KUKA KRL program: MyProgram_171().src

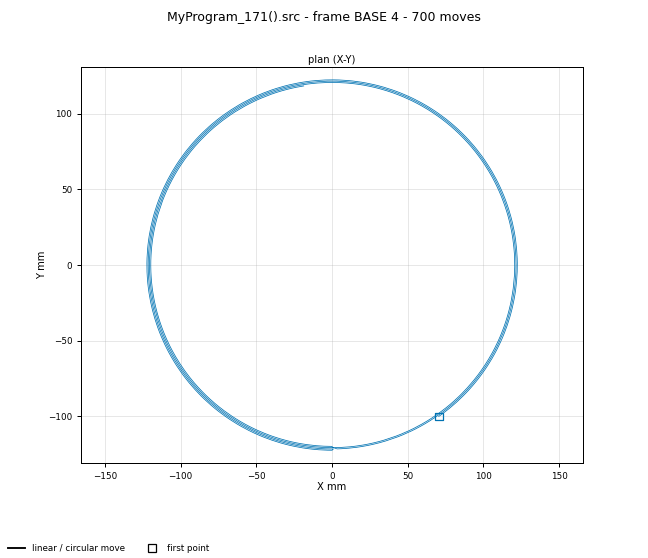
[picture p0: tool path of MyProgram_171().src in frame BASE 4, 700 of 700 moves have a stored position in this frame; points joined in program order, loops and branches not executed]
&ACCESS RVP
&REL 1
&PARAM TEMPLATE = C:\KRC\Roboter\Template\vorgabe
&PARAM EDITMASK = *
DEF MyProgram_171()
; ---- Setting reference (Base) ----
$BASE = BASE_DATA[4]

; --------------------------
; ---- Setting tool (TCP) ----
$TOOL = TOOL_DATA[3]
; --------------------------

$VEL.CP = VEL_APROX_PRINT
Startdeposition()
$VEL.CP = VEL_PRINT
LIN {X 70.4389,Y -100.0155,Z 128,A -58.0013,B 24.9588,C -1.4823,E1 25.0931,E2 504.1944} C_DIS
LIN {X 73.2543,Y -97.9697,Z 128,A -56.5791,B 24.9592,C -1.4754,E1 25.0962,E2 502.7935} C_DIS
LIN {X 75.6365,Y -96.1425,Z 128,A -55.0497,B 24.9587,C -1.4846,E1 25.0997,E2 501.248} C_DIS
LIN {X 77.6056,Y -94.5627,Z 128,A -53.6502,B 24.958,C -1.4981,E1 25.1027,E2 499.822} C_DIS
LIN {X 80.2629,Y -92.3154,Z 128,A -52.1799,B 24.9582,C -1.4939,E1 25.1058,E2 498.3674} C_DIS
LIN {X 82.1521,Y -90.6409,Z 128,A -50.8516,B 24.9576,C -1.504,E1 25.1086,E2 497.0206} C_DIS
LIN {X 84.6959,Y -88.2659,Z 128,A -49.3816,B 24.9579,C -1.4999,E1 25.1116,E2 495.5662} C_DIS
LIN {X 86.5007,Y -86.5007,Z 128,A -48.187,B 24.9577,C -1.5034,E1 25.1139,E2 494.3684} C_DIS
LIN {X 88.5975,Y -84.3518,Z 128,A -46.655,B 24.9571,C -1.5133,E1 25.1169,E2 492.8197} C_DIS
LIN {X 90.6409,Y -82.1521,Z 128,A -45.408,B 24.9573,C -1.5089,E1 25.1192,E2 491.5886} C_DIS
LIN {X 92.6297,Y -79.903,Z 128,A -43.8579,B 24.9567,C -1.5198,E1 25.1221,E2 490.0197} C_DIS
LIN {X 94.8636,Y -77.2344,Z 128,A -42.5892,B 24.9575,C -1.506,E1 25.1243,E2 488.7895} C_DIS
LIN {X 96.7305,Y -74.883,Z 128,A -41.1907,B 24.9573,C -1.5094,E1 25.1267,E2 487.3894} C_DIS
LIN {X 98.5391,Y -72.4866,Z 128,A -39.5927,B 24.9565,C -1.5229,E1 25.1294,E2 485.7672} C_DIS
LIN {X 100.8724,Y -69.2062,Z 128,A -37.5667,B 24.9558,C -1.5353,E1 25.1327,E2 483.7218} C_DIS
LIN {X 102.7986,Y -66.3077,Z 128,A -36.0983,B 24.956,C -1.5318,E1 25.1349,E2 482.269} C_DIS
LIN {X 104.3949,Y -63.7649,Z 128,A -34.9004,B 24.9564,C -1.5254,E1 25.1367,E2 481.0924} C_DIS
LIN {X 105.6902,Y -61.5981,Z 128,A -33.3738,B 24.9552,C -1.5463,E1 25.1389,E2 479.5245} C_DIS
LIN {X 107.3979,Y -58.5657,Z 128,A -31.9057,B 24.9554,C -1.5429,E1 25.1409,E2 478.0719} C_DIS
LIN {X 108.8029,Y -55.9124,Z 128,A -30.7084,B 24.9558,C -1.5366,E1 25.1424,E2 476.8958} C_DIS
LIN {X 110.1423,Y -53.2254,Z 128,A -29.1112,B 24.955,C -1.5505,E1 25.1444,E2 475.2744} C_DIS
LIN {X 111.219,Y -50.942,Z 128,A -27.9364,B 24.9548,C -1.5537,E1 25.1458,E2 474.0984} C_DIS
LIN {X 112.4356,Y -48.1972,Z 128,A -26.3877,B 24.9541,C -1.5653,E1 25.1475,E2 472.5308} C_DIS
LIN {X 113.7054,Y -45.1159,Z 128,A -25.1268,B 24.9547,C -1.555,E1 25.1488,E2 471.3013} C_DIS
LIN {X 114.8289,Y -42.1733,Z 128,A -23.5232,B 24.954,C -1.5661,E1 25.1504,E2 469.6803} C_DIS
LIN {X 115.6766,Y -39.7954,Z 128,A -22.3486,B 24.9538,C -1.5694,E1 25.1515,E2 468.5045} C_DIS
LIN {X 116.7599,Y -36.4881,Z 128,A -20.9292,B 24.9542,C -1.564,E1 25.1527,E2 467.106} C_DIS
LIN {X 117.4899,Y -34.0714,Z 128,A -19.5551,B 24.9534,C -1.5775,E1 25.1538,E2 465.708} C_DIS
LIN {X 118.4097,Y -30.715,Z 128,A -17.9362,B 24.9531,C -1.5822,E1 25.1549,E2 464.0872} C_DIS
LIN {X 119.1278,Y -27.7998,Z 128,A -16.7141,B 24.9534,C -1.5774,E1 25.1557,E2 462.8836} C_DIS
LIN {X 119.7741,Y -24.8679,Z 128,A -15.3426,B 24.9532,C -1.5802,E1 25.1566,E2 461.5134} C_DIS
LIN {X 120.2638,Y -22.3914,Z 128,A -13.9111,B 24.9522,C -1.5966,E1 25.1573,E2 460.0515} C_DIS
LIN {X 120.7771,Y -19.4332,Z 128,A -12.5721,B 24.9522,C -1.5978,E1 25.1579,E2 458.7176} C_DIS
LIN {X 121.2176,Y -16.4633,Z 128,A -11.1755,B 24.9519,C -1.6019,E1 25.1585,E2 457.3195} C_DIS
LIN {X 121.6349,Y -13.0082,Z 128,A -9.7568,B 24.9522,C -1.5966,E1 25.1589,E2 455.9219} C_DIS
LIN {X 121.8794,Y -10.4956,Z 128,A -8.3826,B 24.9514,C -1.6102,E1 25.1593,E2 454.5238} C_DIS
LIN {X 122.1266,Y -7.0242,Z 128,A -6.7638,B 24.9511,C -1.615,E1 25.1596,E2 452.9033} C_DIS
LIN {X 122.2476,Y -4.5026,Z 128,A -5.5896,B 24.9509,C -1.6184,E1 25.1597,E2 451.7279} C_DIS
LIN {X 122.3219,Y -1.3996,Z 128,A -4.203,B 24.9509,C -1.6198,E1 25.1597,E2 450.3464} C_DIS
LIN {X 122.3213,Y 1.5012,Z 128,A -2.645,B 24.9499,C -1.6343,E1 25.1597,E2 448.7633} C_DIS
LIN {X 122.2476,Y 4.5026,Z 128,A -1.4,B 24.9502,C -1.6307,E1 25.1597,E2 447.5342} C_DIS
LIN {X 122.068,Y 7.9782,Z 128,A 0.0188,B 24.9505,C -1.6254,E1 25.1594,E2 446.1364} C_DIS
LIN {X 121.8794,Y 10.4956,Z 128,A 1.5445,B 24.9492,C -1.6466,E1 25.1591,E2 444.5698} C_DIS
LIN {X 121.5295,Y 13.9582,Z 128,A 2.8121,B 24.95,C -1.6335,E1 25.1587,E2 443.3405} C_DIS
LIN {X 121.2176,Y 16.4633,Z 128,A 4.3379,B 24.9487,C -1.6547,E1 25.1581,E2 441.7738} C_DIS
LIN {X 120.7771,Y 19.4332,Z 128,A 5.7347,B 24.9484,C -1.6587,E1 25.1575,E2 440.3757} C_DIS
LIN {X 120.1591,Y 22.935,Z 128,A 7.2165,B 24.9487,C -1.6547,E1 25.1568,E2 438.912} C_DIS
LIN {X 119.5762,Y 25.8029,Z 128,A 8.3989,B 24.949,C -1.6495,E1 25.1561,E2 437.7487} C_DIS
LIN {X 119.0202,Y 28.2654,Z 128,A 9.7736,B 24.9482,C -1.6629,E1 25.1552,E2 436.3504} C_DIS
LIN {X 118.1661,Y 31.6392,Z 128,A 11.393,B 24.9479,C -1.6675,E1 25.1541,E2 434.7296} C_DIS
LIN {X 117.354,Y 34.5296,Z 128,A 12.7898,B 24.9477,C -1.6714,E1 25.153,E2 433.3317} C_DIS
LIN {X 116.6184,Y 36.9445,Z 128,A 13.9648,B 24.9475,C -1.6746,E1 25.152,E2 432.1558} C_DIS
LIN {X 115.6766,Y 39.7954,Z 128,A 15.362,B 24.9472,C -1.6784,E1 25.1508,E2 430.7575} C_DIS
LIN {X 114.4959,Y 43.0691,Z 128,A 16.9816,B 24.9469,C -1.6828,E1 25.1492,E2 429.1365} C_DIS
LIN {X 113.4044,Y 45.866,Z 128,A 18.379,B 24.9467,C -1.6865,E1 25.1478,E2 427.7382} C_DIS
LIN {X 112.2447,Y 48.6353,Z 128,A 19.7766,B 24.9465,C -1.6902,E1 25.1463,E2 426.3395} C_DIS
LIN {X 111.0173,Y 51.3753,Z 128,A 20.9741,B 24.9469,C -1.6838,E1 25.1449,E2 425.1636} C_DIS
LIN {X 109.723,Y 54.0843,Z 128,A 22.5719,B 24.946,C -1.6974,E1 25.1429,E2 423.5423} C_DIS
LIN {X 108.3627,Y 56.7608,Z 128,A 23.9696,B 24.9458,C -1.7009,E1 25.1411,E2 422.1436} C_DIS
LIN {X 106.9371,Y 59.403,Z 128,A 25.3677,B 24.9456,C -1.7044,E1 25.1393,E2 420.7446} C_DIS
LIN {X 105.6902,Y 61.5981,Z 128,A 26.5436,B 24.9454,C -1.7073,E1 25.1376,E2 419.568} C_DIS
LIN {X 103.8935,Y 64.5786,Z 128,A 28.1838,B 24.9451,C -1.7122,E1 25.1352,E2 417.9246} C_DIS
LIN {X 102.2598,Y 67.1355,Z 128,A 29.5683,B 24.9449,C -1.7141,E1 25.1331,E2 416.5425} C_DIS
LIN {X 100.8724,Y 69.2062,Z 128,A 30.7386,B 24.9447,C -1.7173,E1 25.1313,E2 415.3706} C_DIS
LIN {X 99.0399,Y 71.8026,Z 128,A 32.312,B 24.9442,C -1.7253,E1 25.1287,E2 413.7858} C_DIS
LIN {X 97.0634,Y 74.451,Z 128,A 33.5581,B 24.9449,C -1.7142,E1 25.1267,E2 412.5719} C_DIS
LIN {X 95.508,Y 76.4394,Z 128,A 34.9349,B 24.9441,C -1.7267,E1 25.1242,E2 411.1721} C_DIS
LIN {X 93.6033,Y 78.7602,Z 128,A 36.4861,B 24.9434,C -1.7372,E1 25.1214,E2 409.6032} C_DIS
LIN {X 90.6409,Y 82.1521,Z 128,A 38.585,B 24.9432,C -1.7416,E1 25.1175,E2 407.5033} C_DIS
LIN {X 88.2659,Y 84.6959,Z 128,A 40.0554,B 24.9434,C -1.7373,E1 25.1147,E2 406.0493} C_DIS
LIN {X 86.088,Y 86.9084,Z 128,A 41.4744,B 24.9434,C -1.7388,E1 25.112,E2 404.6329} C_DIS
LIN {X 82.9061,Y 89.9491,Z 128,A 43.555,B 24.943,C -1.744,E1 25.1077,E2 402.5484} C_DIS
LIN {X 80.6293,Y 91.9953,Z 128,A 44.9663,B 24.9429,C -1.7458,E1 25.1048,E2 401.1385} C_DIS
LIN {X 77.2344,Y 94.8636,Z 128,A 47.0559,B 24.9426,C -1.7503,E1 25.1003,E2 399.0465} C_DIS
LIN {X 74.883,Y 96.7305,Z 128,A 48.4567,B 24.9424,C -1.7526,E1 25.0972,E2 397.6453} C_DIS
LIN {X 72.4866,Y 98.5391,Z 128,A 49.8576,B 24.9423,C -1.7549,E1 25.0941,E2 396.2442} C_DIS
LIN {X 70.4389,Y 100.0155,Z 128,A 51.188,B 24.9417,C -1.7641,E1 25.091,E2 394.8966} C_DIS
LIN {X 67.5642,Y 101.9771,Z 128,A 52.6957,B 24.9419,C -1.7609,E1 25.0875,E2 393.4015} C_DIS
LIN {X 64.1733,Y 104.1467,Z 128,A 54.5393,B 24.9419,C -1.7618,E1 25.0832,E2 391.5618} C_DIS
LIN {X 61.1837,Y 105.9283,Z 128,A 56.1641,B 24.9417,C -1.764,E1 25.0793,E2 389.9367} C_DIS
LIN {X 58.5657,Y 107.3979,Z 128,A 57.566,B 24.9416,C -1.7657,E1 25.0758,E2 388.5347} C_DIS
LIN {X 55.9124,Y 108.8029,Z 128,A 58.9683,B 24.9415,C -1.7674,E1 25.0724,E2 387.1323} C_DIS
LIN {X 53.6561,Y 109.9353,Z 128,A 60.3,B 24.9409,C -1.7761,E1 25.069,E2 385.7836} C_DIS
LIN {X 50.7212,Y 111.3185,Z 128,A 61.7354,B 24.941,C -1.7738,E1 25.0654,E2 384.3572} C_DIS
LIN {X 47.7569,Y 112.6212,Z 128,A 63.1765,B 24.9412,C -1.7719,E1 25.0617,E2 382.9241} C_DIS
LIN {X 45.4234,Y 113.5846,Z 128,A 64.3564,B 24.9411,C -1.773,E1 25.0586,E2 381.7444} C_DIS
LIN {X 42.6222,Y 114.6651,Z 128,A 65.7597,B 24.9411,C -1.7742,E1 25.055,E2 380.3412} C_DIS
LIN {X 39.7954,Y 115.6766,Z 128,A 67.3158,B 24.9404,C -1.7826,E1 25.0508,E2 378.7683} C_DIS
LIN {X 36.4881,Y 116.7599,Z 128,A 68.664,B 24.9412,C -1.7705,E1 25.0473,E2 377.4512} C_DIS
LIN {X 34.0714,Y 117.4899,Z 128,A 69.9711,B 24.9408,C -1.7773,E1 25.0438,E2 376.1304} C_DIS
LIN {X 30.715,Y 118.4097,Z 128,A 71.3977,B 24.9414,C -1.7688,E1 25.04,E2 374.7263} C_DIS
LIN {X 27.7998,Y 119.1278,Z 128,A 72.8019,B 24.9414,C -1.7695,E1 25.0362,E2 373.3224} C_DIS
LIN {X 24.8679,Y 119.7741,Z 128,A 74.4081,B 24.9406,C -1.7796,E1 25.0318,E2 371.6942} C_DIS
LIN {X 22.3914,Y 120.2638,Z 128,A 75.5897,B 24.9406,C -1.7801,E1 25.0285,E2 370.513} C_DIS
LIN {X 19.4332,Y 120.7771,Z 128,A 76.9948,B 24.9406,C -1.7805,E1 25.0246,E2 369.1083} C_DIS
LIN {X 15.9894,Y 121.279,Z 128,A 78.4225,B 24.9412,C -1.7714,E1 25.0208,E2 367.7033} C_DIS
LIN {X 13.4835,Y 121.5851,Z 128,A 79.9588,B 24.9401,C -1.7882,E1 25.0164,E2 366.1283} C_DIS
LIN {X 10.1865,Y 121.9041,Z 128,A 81.356,B 24.9405,C -1.7812,E1 25.0126,E2 364.7487} C_DIS
LIN {X 7.0242,Y 122.1266,Z 128,A 82.8419,B 24.9405,C -1.7812,E1 25.0084,E2 363.2632} C_DIS
LIN {X 4.5026,Y 122.2476,Z 128,A 84.0246,B 24.9405,C -1.7812,E1 25.0051,E2 362.0811} C_DIS
LIN {X 1.0233,Y 122.3242,Z 128,A 85.4534,B 24.9412,C -1.7716,E1 25.0012,E2 360.6751} C_DIS
LIN {X -1.979,Y 122.3125,Z 128,A 87.0621,B 24.9406,C -1.7807,E1 24.9966,E2 359.0449} C_DIS
LIN {X -4.5026,Y 122.2476,Z 128,A 88.2453,B 24.9406,C -1.7803,E1 24.9933,E2 357.8624} C_DIS
LIN {X -7.9782,Y 122.068,Z 128,A 89.8768,B 24.9406,C -1.7798,E1 24.9888,E2 356.2317} C_DIS
LIN {X -10.4956,Y 121.8794,Z 128,A 91.0602,B 24.9406,C -1.7792,E1 24.9855,E2 355.049} C_DIS
LIN {X -13.9582,Y 121.5295,Z 128,A 92.5486,B 24.9412,C -1.7719,E1 24.9814,E2 353.5772} C_DIS
LIN {X -16.9365,Y 121.1504,Z 128,A 94.1004,B 24.9408,C -1.7777,E1 24.9771,E2 352.0104} C_DIS
LIN {X -19.9045,Y 120.6982,Z 128,A 95.5087,B 24.9408,C -1.7768,E1 24.9732,E2 350.603} C_DIS
LIN {X -22.8606,Y 120.1734,Z 128,A 96.7156,B 24.9415,C -1.7666,E1 24.9699,E2 349.4191} C_DIS
LIN {X -25.803,Y 119.5762,Z 128,A 98.2874,B 24.9411,C -1.7729,E1 24.9656,E2 347.8304} C_DIS
LIN {X -28.2654,Y 119.0202,Z 128,A 99.511,B 24.9411,C -1.7737,E1 24.9623,E2 346.6033} C_DIS
LIN {X -31.6392,Y 118.1661,Z 128,A 101.1446,B 24.9411,C -1.7722,E1 24.9578,E2 344.9708} C_DIS
LIN {X -34.5296,Y 117.354,Z 128,A 102.352,B 24.9418,C -1.7616,E1 24.9547,E2 343.7866} C_DIS
LIN {X -36.9445,Y 116.6184,Z 128,A 103.8928,B 24.9408,C -1.7766,E1 24.9505,E2 342.2076} C_DIS
LIN {X -39.7954,Y 115.6766,Z 128,A 105.1493,B 24.9414,C -1.768,E1 24.9472,E2 340.9692} C_DIS
LIN {X -43.0691,Y 114.4959,Z 128,A 106.7841,B 24.9415,C -1.7661,E1 24.9429,E2 339.3355} C_DIS
LIN {X -45.4234,Y 113.5846,Z 128,A 108.1235,B 24.9412,C -1.7715,E1 24.9394,E2 337.9803} C_DIS
LIN {X -48.6353,Y 112.2447,Z 128,A 109.6052,B 24.9418,C -1.7625,E1 24.9356,E2 336.5167} C_DIS
LIN {X -51.3753,Y 111.0173,Z 128,A 111.0161,B 24.9419,C -1.7605,E1 24.932,E2 335.1069} C_DIS
LIN {X -53.6561,Y 109.9353,Z 128,A 112.2025,B 24.942,C -1.7588,E1 24.9291,E2 333.9216} C_DIS
LIN {X -56.7608,Y 108.3627,Z 128,A 113.6359,B 24.9428,C -1.7473,E1 24.9256,E2 332.5117} C_DIS
LIN {X -58.9858,Y 107.1701,Z 128,A 115.1787,B 24.9419,C -1.7614,E1 24.9217,E2 330.931} C_DIS
LIN {X -61.5981,Y 105.6902,Z 128,A 116.5984,B 24.9419,C -1.7594,E1 24.9183,E2 329.5116} C_DIS
LIN {X -64.2066,Y 104.1259,Z 128,A 117.8506,B 24.9427,C -1.749,E1 24.9153,E2 328.2804} C_DIS
LIN {X -66.7099,Y 102.5404,Z 128,A 119.2609,B 24.9427,C -1.7474,E1 24.912,E2 326.8695} C_DIS
LIN {X -69.5986,Y 100.5996,Z 128,A 120.6954,B 24.9436,C -1.7354,E1 24.9087,E2 325.4586} C_DIS
LIN {X -71.6609,Y 99.1436,Z 128,A 122.0858,B 24.9431,C -1.7422,E1 24.9055,E2 324.0472} C_DIS
LIN {X -74.0725,Y 97.3551,Z 128,A 123.4985,B 24.9433,C -1.7395,E1 24.9024,E2 322.6359} C_DIS
LIN {X -76.4394,Y 95.508,Z 128,A 125.0647,B 24.943,C -1.7436,E1 24.8989,E2 321.0542} C_DIS
LIN {X -79.124,Y 93.2934,Z 128,A 126.549,B 24.9437,C -1.7334,E1 24.8958,E2 319.5883} C_DIS
LIN {X -81.3897,Y 91.3235,Z 128,A 127.7595,B 24.9445,C -1.7215,E1 24.8933,E2 318.4013} C_DIS
LIN {X -83.6064,Y 89.2986,Z 128,A 129.1729,B 24.9447,C -1.7185,E1 24.8904,E2 316.9894} C_DIS
LIN {X -85.4327,Y 87.5557,Z 128,A 130.7185,B 24.9438,C -1.7317,E1 24.8872,E2 315.406} C_DIS
LIN {X -87.5735,Y 85.4142,Z 128,A 131.979,B 24.9445,C -1.7212,E1 24.8848,E2 314.1651} C_DIS
LIN {X -89.9491,Y 82.9061,Z 128,A 133.6167,B 24.9447,C -1.718,E1 24.8817,E2 312.5278} C_DIS
LIN {X -91.9566,Y 80.6737,Z 128,A 135.0309,B 24.9449,C -1.7148,E1 24.879,E2 311.1151} C_DIS
LIN {X -93.9087,Y 78.3927,Z 128,A 136.445,B 24.9451,C -1.7114,E1 24.8765,E2 309.7024} C_DIS
LIN {X -95.7506,Y 76.1323,Z 128,A 137.6524,B 24.9458,C -1.7008,E1 24.8744,E2 308.5146} C_DIS
LIN {X -97.4209,Y 73.9849,Z 128,A 139.2166,B 24.9452,C -1.7101,E1 24.8717,E2 306.9209} C_DIS
LIN {X -99.4212,Y 71.2719,Z 128,A 140.6881,B 24.9458,C -1.701,E1 24.8693,E2 305.4638} C_DIS
LIN {X -100.8724,Y 69.2062,Z 128,A 141.8779,B 24.946,C -1.698,E1 24.8674,E2 304.2753} C_DIS
LIN {X -102.7986,Y 66.3077,Z 128,A 143.315,B 24.9468,C -1.685,E1 24.8653,E2 302.8621} C_DIS
LIN {X -104.3949,Y 63.7649,Z 128,A 144.9327,B 24.9465,C -1.6902,E1 24.8628,E2 301.2238} C_DIS
LIN {X -105.6902,Y 61.5981,Z 128,A 146.1228,B 24.9467,C -1.687,E1 24.8612,E2 300.035} C_DIS
LIN {X -107.3979,Y 58.5657,Z 128,A 147.7629,B 24.9469,C -1.6827,E1 24.8589,E2 298.3967} C_DIS
LIN {X -108.5854,Y 56.3379,Z 128,A 148.9532,B 24.9471,C -1.6795,E1 24.8574,E2 297.2077} C_DIS
LIN {X -110.1423,Y 53.2254,Z 128,A 150.3908,B 24.948,C -1.6662,E1 24.8556,E2 295.794} C_DIS
LIN {X -111.219,Y 50.942,Z 128,A 151.7839,B 24.9476,C -1.6717,E1 24.854,E2 294.3801} C_DIS
LIN {X -112.4356,Y 48.1972,Z 128,A 153.1996,B 24.9479,C -1.6678,E1 24.8524,E2 292.9659} C_DIS
LIN {X -113.5846,Y 45.4234,Z 128,A 154.6152,B 24.9481,C -1.6638,E1 24.8509,E2 291.5519} C_DIS
LIN {X -114.6651,Y 42.6222,Z 128,A 156.0308,B 24.9484,C -1.6599,E1 24.8495,E2 290.1377} C_DIS
LIN {X -115.8293,Y 39.3425,Z 128,A 157.6716,B 24.9487,C -1.6552,E1 24.848,E2 288.4987} C_DIS
LIN {X -116.7599,Y 36.4881,Z 128,A 158.8849,B 24.9495,C -1.6424,E1 24.847,E2 287.3091} C_DIS
LIN {X -117.4899,Y 34.0714,Z 128,A 160.2783,B 24.9491,C -1.6477,E1 24.8459,E2 285.8948} C_DIS
LIN {X -118.4097,Y 30.715,Z 128,A 161.7167,B 24.95,C -1.6342,E1 24.8448,E2 284.4803} C_DIS
LIN {X -119.1278,Y 27.7998,Z 128,A 163.1324,B 24.9502,C -1.6301,E1 24.8439,E2 283.0662} C_DIS
LIN {X -119.7144,Y 25.1591,Z 128,A 164.5349,B 24.9502,C -1.6318,E1 24.8431,E2 281.6513} C_DIS
LIN {X -120.2638,Y 22.3914,Z 128,A 165.9425,B 24.9502,C -1.6313,E1 24.8423,E2 280.2367} C_DIS
LIN {X -120.7771,Y 19.4332,Z 128,A 167.5124,B 24.95,C -1.6338,E1 24.8416,E2 278.6513} C_DIS
LIN {X -121.279,Y 15.9894,Z 128,A 168.7971,B 24.9512,C -1.6135,E1 24.8411,E2 277.4074} C_DIS
LIN {X -121.6349,Y 13.0082,Z 128,A 170.4159,B 24.9509,C -1.6181,E1 24.8406,E2 275.7679} C_DIS
LIN {X -121.9175,Y 10.0192,Z 128,A 171.8018,B 24.9513,C -1.6127,E1 24.8403,E2 274.3868} C_DIS
LIN {X -122.1266,Y 7.0242,Z 128,A 173.2484,B 24.9514,C -1.6098,E1 24.84,E2 272.9382} C_DIS
LIN {X -122.2476,Y 4.5026,Z 128,A 174.4392,B 24.9517,C -1.6063,E1 24.8399,E2 271.7487} C_DIS
LIN {X -122.3233,Y 1.1863,Z 128,A 176.0133,B 24.9519,C -1.6021,E1 24.8398,E2 270.175} C_DIS
LIN {X -122.3125,Y -1.979,Z 128,A 177.4968,B 24.9522,C -1.5973,E1 24.8398,E2 268.694} C_DIS
LIN {X -122.2476,Y -4.5026,Z 128,A 178.6875,B 24.9524,C -1.5938,E1 24.8399,E2 267.5045} C_DIS
LIN {X -122.068,Y -7.9782,Z 128,A -179.6453,B 24.9526,C -1.5901,E1 24.8402,E2 265.836} C_DIS
LIN {X -121.7414,Y -11.9905,Z 128,A -177.6185,B 24.9526,C -1.5901,E1 24.8407,E2 263.797} C_DIS
LIN {X -121.3491,Y -15.4485,Z 128,A -176.1313,B 24.9533,C -1.5787,E1 24.8412,E2 262.3282} C_DIS
LIN {X -120.9334,Y -18.4219,Z 128,A -174.7152,B 24.9535,C -1.5747,E1 24.8418,E2 260.9134} C_DIS
LIN {X -120.4449,Y -21.3842,Z 128,A -173.2995,B 24.9538,C -1.5706,E1 24.8425,E2 259.4989} C_DIS
LIN {X -119.8927,Y -24.2902,Z 128,A -171.8914,B 24.954,C -1.5672,E1 24.8432,E2 258.0906} C_DIS
LIN {X -119.3581,Y -26.8028,Z 128,A -170.693,B 24.9542,C -1.5632,E1 24.8439,E2 256.8947} C_DIS
LIN {X -118.6644,Y -29.7239,Z 128,A -169.1237,B 24.9541,C -1.5659,E1 24.845,E2 255.3096} C_DIS
LIN {X -117.7689,Y -33.0869,Z 128,A -167.6366,B 24.9547,C -1.5547,E1 24.8461,E2 253.8408} C_DIS
LIN {X -117.063,Y -35.5107,Z 128,A -166.2925,B 24.9545,C -1.5581,E1 24.8472,E2 252.4808} C_DIS
LIN {X -116.0035,Y -38.8257,Z 128,A -165.0085,B 24.9557,C -1.538,E1 24.8482,E2 251.2373} C_DIS
LIN {X -115.1795,Y -41.2119,Z 128,A -163.4617,B 24.955,C -1.5504,E1 24.8497,E2 249.6521} C_DIS
LIN {X -113.9587,Y -44.4709,Z 128,A -162.1781,B 24.9561,C -1.5303,E1 24.8509,E2 248.4091} C_DIS
LIN {X -112.833,Y -47.2542,Z 128,A -160.5601,B 24.9558,C -1.5355,E1 24.8527,E2 246.7698} C_DIS
LIN {X -111.6394,Y -50.0091,Z 128,A -159.3475,B 24.9565,C -1.5229,E1 24.854,E2 245.5806} C_DIS
LIN {X -110.5854,Y -52.303,Z 128,A -157.8015,B 24.9558,C -1.5355,E1 24.8559,E2 243.996} C_DIS
LIN {X -109.2686,Y -55.0012,Z 128,A -156.5402,B 24.9564,C -1.5251,E1 24.8574,E2 242.7528} C_DIS
LIN {X -107.8859,Y -57.6662,Z 128,A -155.1256,B 24.9566,C -1.5216,E1 24.8593,E2 241.3391} C_DIS
LIN {X -106.2001,Y -60.7108,Z 128,A -153.4379,B 24.9567,C -1.5197,E1 24.8616,E2 239.6471} C_DIS
LIN {X -104.1467,Y -64.1733,Z 128,A -151.5897,B 24.9571,C -1.5129,E1 24.8643,E2 237.8054} C_DIS
LIN {X -102.5404,Y -66.7099,Z 128,A -150.022,B 24.9569,C -1.5164,E1 24.8666,E2 236.2214} C_DIS
LIN {X -100.5996,Y -69.5986,Z 128,A -148.7391,B 24.958,C -1.4968,E1 24.8686,E2 234.9789} C_DIS
LIN {X -99.1436,Y -71.6609,Z 128,A -147.1939,B 24.9573,C -1.51,E1 24.8712,E2 233.3949} C_DIS
LIN {X -97.0201,Y -74.5073,Z 128,A -145.6955,B 24.9579,C -1.4985,E1 24.8737,E2 231.9165} C_DIS
LIN {X -94.5627,Y -77.6056,Z 128,A -143.66,B 24.9577,C -1.5022,E1 24.8773,E2 229.8627} C_DIS
LIN {X -92.3154,Y -80.2629,Z 128,A -142.1753,B 24.9583,C -1.4919,E1 24.8799,E2 228.3958} C_DIS
LIN {X -90.6409,Y -82.1521,Z 128,A -140.8336,B 24.9581,C -1.4964,E1 24.8825,E2 227.0376} C_DIS
LIN {X -88.2659,Y -84.6959,Z 128,A -139.3492,B 24.9586,C -1.4862,E1 24.8853,E2 225.5708} C_DIS
LIN {X -86.5007,Y -86.5007,Z 128,A -138.1613,B 24.9587,C -1.4839,E1 24.8876,E2 224.3834} C_DIS
LIN {X -84.3518,Y -88.5975,Z 128,A -136.5954,B 24.9585,C -1.4881,E1 24.8908,E2 222.8009} C_DIS
LIN {X -81.8156,Y -90.9422,Z 128,A -135.315,B 24.9595,C -1.4696,E1 24.8934,E2 221.5594} C_DIS
LIN {X -79.903,Y -92.6297,Z 128,A -133.7708,B 24.9588,C -1.4831,E1 24.8967,E2 219.9772} C_DIS
LIN {X -77.2344,Y -94.8636,Z 128,A -132.4901,B 24.9598,C -1.4641,E1 24.8994,E2 218.7366} C_DIS
LIN {X -74.883,Y -96.7305,Z 128,A -130.8258,B 24.9593,C -1.4733,E1 24.9031,E2 217.0445} C_DIS
LIN {X -72.4866,Y -98.5391,Z 128,A -129.4643,B 24.9596,C -1.4687,E1 24.9061,E2 215.6889} C_DIS
LIN {X -70.4389,Y -100.0155,Z 128,A -128.2773,B 24.9596,C -1.4669,E1 24.9088,E2 214.5022} C_DIS
LIN {X -67.5642,Y -101.9771,Z 128,A -126.6415,B 24.9598,C -1.4645,E1 24.9126,E2 212.8667} C_DIS
LIN {X -65.0412,Y -103.6045,Z 128,A -125.2306,B 24.9599,C -1.4625,E1 24.9159,E2 211.4559} C_DIS
LIN {X -62.8904,Y -104.9264,Z 128,A -124.0444,B 24.96,C -1.4609,E1 24.9188,E2 210.2699} C_DIS
LIN {X -59.8792,Y -106.6712,Z 128,A -122.4094,B 24.9601,C -1.4588,E1 24.9227,E2 208.6351} C_DIS
LIN {X -57.2434,Y -108.1085,Z 128,A -120.9991,B 24.9602,C -1.4571,E1 24.9262,E2 207.2248} C_DIS
LIN {X -55.0012,Y -109.2686,Z 128,A -119.6604,B 24.9599,C -1.4628,E1 24.9296,E2 205.869} C_DIS
LIN {X -51.8698,Y -110.7871,Z 128,A -118.1491,B 24.9603,C -1.4554,E1 24.9334,E2 204.3715} C_DIS
LIN {X -48.1972,Y -112.4356,Z 128,A -116.1362,B 24.9601,C -1.4592,E1 24.9385,E2 202.3448} C_DIS
LIN {X -45.4234,Y -113.5846,Z 128,A -114.7346,B 24.9602,C -1.4575,E1 24.9422,E2 200.9441} C_DIS
LIN {X -42.1733,Y -114.8289,Z 128,A -113.2466,B 24.9606,C -1.4494,E1 24.946,E2 199.4722} C_DIS
LIN {X -39.7954,Y -115.6766,Z 128,A -112.0563,B 24.9606,C -1.4488,E1 24.9492,E2 198.2812} C_DIS
LIN {X -36.4881,Y -116.7599,Z 128,A -110.6306,B 24.9613,C -1.438,E1 24.9529,E2 196.8785} C_DIS
LIN {X -34.0714,Y -117.4899,Z 128,A -109.2449,B 24.9608,C -1.4466,E1 24.9567,E2 195.47} C_DIS
LIN {X -30.715,Y -118.4097,Z 128,A -107.6128,B 24.9608,C -1.4457,E1 24.9611,E2 193.8375} C_DIS
LIN {X -27.7998,Y -119.1278,Z 128,A -106.4066,B 24.9614,C -1.4356,E1 24.9643,E2 192.6537} C_DIS
LIN {X -24.8679,Y -119.7741,Z 128,A -104.9985,B 24.9614,C -1.435,E1 24.9681,E2 191.2453} C_DIS
LIN {X -21.906,Y -120.3511,Z 128,A -103.5905,B 24.9614,C -1.4342,E1 24.972,E2 189.8377} C_DIS
LIN {X -19.4332,Y -120.7771,Z 128,A -102.2066,B 24.961,C -1.4436,E1 24.9759,E2 188.4301} C_DIS
LIN {X -16.4633,Y -121.2176,Z 128,A -100.7996,B 24.961,C -1.4433,E1 24.9798,E2 187.0227} C_DIS
LIN {X -13.0082,Y -121.6349,Z 128,A -99.1438,B 24.961,C -1.4443,E1 24.9844,E2 185.3633} C_DIS
LIN {X -8.9992,Y -121.999,Z 128,A -97.1309,B 24.9606,C -1.4503,E1 24.99,E2 183.3354} C_DIS
LIN {X -5.525,Y -122.2036,Z 128,A -95.8548,B 24.9615,C -1.4336,E1 24.9935,E2 182.0986} C_DIS
LIN {X -3.0021,Y -122.2936,Z 128,A -94.3189,B 24.9606,C -1.4506,E1 24.9979,E2 180.5223} C_DIS
LIN {X 0,Y -122.3305,Z 128,A -92.9133,B 24.9606,C -1.4508,E1 25.0018,E2 179.1161} C_DIS
LIN {X 0,Y -122.3305,Z 128,A -92.9133,B 24.9606,C -1.4508,E1 25.0018,E2 179.1161} C_DIS
Enddeposition()
LIN {X 0.8564,Y -121.47,Z 128,A -92.5769,B 24.9599,C -1.4627,E1 25.0028,E2 178.7516} C_DIS
Startdeposition()
$VEL.CP = VEL_PRINT
LIN {X -0.9647,Y -121.4729,Z 128,A -94.2168,B 24.9619,C -1.4256,E1 24.998,E2 180.4793} C_DIS
LIN {X -4.555,Y -121.3929,Z 128,A -96.0357,B 24.9623,C -1.4195,E1 24.9929,E2 182.3129} C_DIS
LIN {X -9.0533,Y -121.1404,Z 128,A -98.2299,B 24.9624,C -1.4163,E1 24.9867,E2 184.5156} C_DIS
LIN {X -13.6853,Y -120.7041,Z 128,A -100.2672,B 24.962,C -1.4238,E1 24.9811,E2 186.5362} C_DIS
LIN {X -17.9499,Y -120.1444,Z 128,A -102.1563,B 24.9617,C -1.4307,E1 24.9759,E2 188.4105} C_DIS
LIN {X -23.0019,Y -119.279,Z 128,A -104.5486,B 24.9616,C -1.4326,E1 24.9694,E2 190.8004} C_DIS
LIN {X -25.7925,Y -118.7068,Z 128,A -106.0689,B 24.962,C -1.4251,E1 24.9651,E2 192.3404} C_DIS
LIN {X -29.1299,Y -117.9327,Z 128,A -107.5553,B 24.9616,C -1.4319,E1 24.9611,E2 193.8127} C_DIS
LIN {X -32.1278,Y -117.1519,Z 128,A -109.0894,B 24.9617,C -1.4295,E1 24.957,E2 195.3549} C_DIS
LIN {X -35.8702,Y -116.0599,Z 128,A -111.0253,B 24.9619,C -1.4263,E1 24.9518,E2 197.3015} C_DIS
LIN {X -38.6924,Y -115.1498,Z 128,A -112.4178,B 24.9619,C -1.4277,E1 24.9481,E2 198.6933} C_DIS
LIN {X -41.7788,Y -114.0663,Z 128,A -113.9264,B 24.9617,C -1.4307,E1 24.9441,E2 200.1979} C_DIS
LIN {X -45.5578,Y -112.6104,Z 128,A -115.8907,B 24.9617,C -1.4301,E1 24.939,E2 202.1678} C_DIS
LIN {X -49.3374,Y -111.008,Z 128,A -117.8037,B 24.9615,C -1.4332,E1 24.9341,E2 204.0778} C_DIS
LIN {X -52.4934,Y -109.5491,Z 128,A -119.3831,B 24.9613,C -1.4379,E1 24.9301,E2 205.6501} C_DIS
LIN {X -55.8126,Y -107.8975,Z 128,A -121.103,B 24.9611,C -1.4414,E1 24.9259,E2 207.3663} C_DIS
LIN {X -58.0544,Y -106.7064,Z 128,A -122.3071,B 24.9611,C -1.4428,E1 24.9229,E2 208.5706} C_DIS
LIN {X -60.7675,Y -105.1853,Z 128,A -123.8443,B 24.9611,C -1.4417,E1 24.9192,E2 210.1148} C_DIS
LIN {X -63.5715,Y -103.5159,Z 128,A -125.3187,B 24.9608,C -1.4469,E1 24.9156,E2 211.5815} C_DIS
LIN {X -66.1342,Y -101.898,Z 128,A -126.9367,B 24.9611,C -1.4407,E1 24.9118,E2 213.2194} C_DIS
LIN {X -69.9741,Y -99.301,Z 128,A -129.1106,B 24.9609,C -1.4449,E1 24.9068,E2 215.3906} C_DIS
LIN {X -73.0883,Y -97.0293,Z 128,A -130.7953,B 24.9604,C -1.4541,E1 24.9031,E2 217.0595} C_DIS
LIN {X -75.5152,Y -95.1529,Z 128,A -132.2867,B 24.9604,C -1.4547,E1 24.8998,E2 218.5548} C_DIS
LIN {X -78.2157,Y -92.9481,Z 128,A -133.8764,B 24.9601,C -1.4603,E1 24.8964,E2 220.1375} C_DIS
LIN {X -80.0842,Y -91.3407,Z 128,A -135.0356,B 24.9599,C -1.4627,E1 24.8939,E2 221.2953} C_DIS
LIN {X -82.2674,Y -89.3794,Z 128,A -136.5698,B 24.9601,C -1.4589,E1 24.8907,E2 222.8447} C_DIS
LIN {X -85.0049,Y -86.7813,Z 128,A -138.4181,B 24.9601,C -1.4597,E1 24.887,E2 224.699} C_DIS
LIN {X -87.6266,Y -84.132,Z 128,A -140.0981,B 24.9597,C -1.467,E1 24.8838,E2 226.3688} C_DIS
LIN {X -90.1201,Y -81.4571,Z 128,A -141.87,B 24.9596,C -1.4688,E1 24.8804,E2 228.1443} C_DIS
LIN {X -92.7192,Y -78.4848,Z 128,A -143.6139,B 24.9591,C -1.4783,E1 24.8772,E2 229.8734} C_DIS
LIN {X -94.7059,Y -76.0765,Z 128,A -145.0772,B 24.9588,C -1.4822,E1 24.8747,E2 231.3341} C_DIS
LIN {X -96.9086,Y -73.2489,Z 128,A -146.9191,B 24.959,C -1.4798,E1 24.8715,E2 233.1907} C_DIS
LIN {X -99.1588,Y -70.1734,Z 128,A -148.6115,B 24.9585,C -1.4889,E1 24.8688,E2 234.8697} C_DIS
LIN {X -100.9336,Y -67.597,Z 128,A -150.0543,B 24.9582,C -1.4941,E1 24.8665,E2 236.3071} C_DIS
LIN {X -102.5688,Y -65.0891,Z 128,A -151.4782,B 24.958,C -1.4973,E1 24.8644,E2 237.7306} C_DIS
LIN {X -104.2177,Y -62.4157,Z 128,A -153.2269,B 24.9584,C -1.4897,E1 24.8618,E2 239.5065} C_DIS
LIN {X -106.4782,Y -58.4752,Z 128,A -155.2855,B 24.9579,C -1.4992,E1 24.859,E2 241.5532} C_DIS
LIN {X -108.1197,Y -55.3778,Z 128,A -156.8253,B 24.9574,C -1.5087,E1 24.857,E2 243.0784} C_DIS
LIN {X -109.5034,Y -52.5887,Z 128,A -158.3584,B 24.9573,C -1.5101,E1 24.8551,E2 244.6165} C_DIS
LIN {X -110.8398,Y -49.7106,Z 128,A -159.8436,B 24.957,C -1.5149,E1 24.8534,E2 246.0985} C_DIS
LIN {X -112.4607,Y -45.9256,Z 128,A -161.7733,B 24.9566,C -1.5211,E1 24.8513,E2 248.024} C_DIS
LIN {X -113.6259,Y -42.9618,Z 128,A -163.4959,B 24.9569,C -1.5161,E1 24.8496,E2 249.7682} C_DIS
LIN {X -114.9148,Y -39.3893,Z 128,A -165.2066,B 24.9564,C -1.525,E1 24.848,E2 251.4676} C_DIS
LIN {X -116.068,Y -35.8442,Z 128,A -166.8746,B 24.9559,C -1.5342,E1 24.8466,E2 253.1231} C_DIS
LIN {X -116.9478,Y -32.8609,Z 128,A -168.5712,B 24.9562,C -1.5289,E1 24.8453,E2 254.8423} C_DIS
LIN {X -117.9614,Y -29.0123,Z 128,A -170.2234,B 24.9553,C -1.5444,E1 24.8442,E2 256.4672} C_DIS
LIN {X -118.6984,Y -25.831,Z 128,A -171.7654,B 24.955,C -1.5491,E1 24.8433,E2 258.0069} C_DIS
LIN {X -119.4275,Y -22.2279,Z 128,A -173.4713,B 24.9547,C -1.5558,E1 24.8423,E2 259.707} C_DIS
LIN {X -119.8705,Y -19.6908,Z 128,A -174.8571,B 24.9548,C -1.5524,E1 24.8417,E2 261.1092} C_DIS
LIN {X -120.4702,Y -15.6044,Z 128,A -176.6949,B 24.9542,C -1.5633,E1 24.841,E2 262.9319} C_DIS
LIN {X -120.8293,Y -12.5236,Z 128,A -178.1645,B 24.9539,C -1.5677,E1 24.8405,E2 264.3998} C_DIS
LIN {X -121.1484,Y -8.9531,Z 128,A 179.9828,B 24.954,C -1.5663,E1 24.8401,E2 266.2671} C_DIS
LIN {X -121.367,Y -5.1596,Z 128,A 178.3084,B 24.9534,C -1.5772,E1 24.8399,E2 267.9256} C_DIS
LIN {X -121.4616,Y -1.9319,Z 128,A 176.827,B 24.953,C -1.5839,E1 24.8398,E2 269.3998} C_DIS
LIN {X -121.4737,Y 0.8721,Z 128,A 175.4506,B 24.9529,C -1.5859,E1 24.8398,E2 270.7797} C_DIS
LIN {X -121.3942,Y 4.5248,Z 128,A 173.584,B 24.9529,C -1.5854,E1 24.84,E2 272.6587} C_DIS
LIN {X -121.2009,Y 8.1796,Z 128,A 171.9423,B 24.9523,C -1.5947,E1 24.8402,E2 274.2882} C_DIS
LIN {X -120.9642,Y 11.1457,Z 128,A 170.5873,B 24.952,C -1.6014,E1 24.8406,E2 275.6355} C_DIS
LIN {X -120.6256,Y 14.3549,Z 128,A 169.0419,B 24.9517,C -1.6053,E1 24.841,E2 277.1807} C_DIS
LIN {X -120.2475,Y 17.2368,Z 128,A 167.6268,B 24.9516,C -1.6079,E1 24.8416,E2 278.598} C_DIS
LIN {X -119.6264,Y 21.1241,Z 128,A 165.7103,B 24.9513,C -1.6114,E1 24.8425,E2 280.5175} C_DIS
LIN {X -118.9252,Y 24.7684,Z 128,A 163.8807,B 24.9513,C -1.6138,E1 24.8435,E2 282.3524} C_DIS
LIN {X -118.0544,Y 28.6313,Z 128,A 162.0982,B 24.9506,C -1.6234,E1 24.8446,E2 284.1223} C_DIS
LIN {X -116.851,Y 33.2026,Z 128,A 159.9062,B 24.9501,C -1.6321,E1 24.8462,E2 286.3063} C_DIS
LIN {X -115.9781,Y 36.1341,Z 128,A 158.4638,B 24.9498,C -1.6368,E1 24.8474,E2 287.746} C_DIS
LIN {X -115.0326,Y 39.0398,Z 128,A 156.9917,B 24.9496,C -1.64,E1 24.8487,E2 289.2188} C_DIS
LIN {X -114.119,Y 41.6342,Z 128,A 155.3481,B 24.9503,C -1.6294,E1 24.8503,E2 290.897} C_DIS
LIN {X -112.7939,Y 45.1072,Z 128,A 153.7693,B 24.9495,C -1.6421,E1 24.8519,E2 292.4542} C_DIS
LIN {X -111.2941,Y 48.6848,Z 128,A 152.1337,B 24.9486,C -1.6561,E1 24.8536,E2 294.0656} C_DIS
LIN {X -109.4507,Y 52.6982,Z 128,A 150.2352,B 24.9477,C -1.6703,E1 24.8558,E2 295.9405} C_DIS
LIN {X -108.2071,Y 55.2068,Z 128,A 148.6355,B 24.9482,C -1.6624,E1 24.8579,E2 297.5678} C_DIS
LIN {X -106.4985,Y 58.4379,Z 128,A 146.6386,B 24.9486,C -1.6558,E1 24.8605,E2 299.5909} C_DIS
LIN {X -103.9115,Y 62.9206,Z 128,A 144.4485,B 24.9475,C -1.6737,E1 24.8636,E2 301.7498} C_DIS
LIN {X -102.2054,Y 65.6552,Z 128,A 142.9104,B 24.9473,C -1.6773,E1 24.8659,E2 303.2872} C_DIS
LIN {X -100.5475,Y 68.1671,Z 128,A 141.4494,B 24.9471,C -1.6795,E1 24.8682,E2 304.7502} C_DIS
LIN {X -98.1193,Y 71.6183,Z 128,A 139.4822,B 24.9467,C -1.686,E1 24.8713,E2 306.7114} C_DIS
LIN {X -95.6681,Y 74.8633,Z 128,A 137.4676,B 24.9467,C -1.687,E1 24.8748,E2 308.7332} C_DIS
LIN {X -93.2225,Y 77.886,Z 128,A 135.7117,B 24.9461,C -1.6953,E1 24.8779,E2 310.4776} C_DIS
LIN {X -90.5284,Y 81.0011,Z 128,A 133.7363,B 24.9459,C -1.6989,E1 24.8815,E2 312.4533} C_DIS
LIN {X -87.9513,Y 83.7951,Z 128,A 132.0141,B 24.9454,C -1.7064,E1 24.8848,E2 314.165} C_DIS
LIN {X -85.4098,Y 86.3813,Z 128,A 130.2688,B 24.9453,C -1.7091,E1 24.8882,E2 315.9113} C_DIS
LIN {X -82.6608,Y 89.0184,Z 128,A 128.3308,B 24.9453,C -1.7073,E1 24.8922,E2 317.8617} C_DIS
LIN {X -79.9136,Y 91.4898,Z 128,A 126.672,B 24.9449,C -1.715,E1 24.8956,E2 319.5087} C_DIS
LIN {X -77.1409,Y 93.8416,Z 128,A 124.8428,B 24.9449,C -1.7139,E1 24.8996,E2 321.3477} C_DIS
LIN {X -74.7515,Y 95.7563,Z 128,A 123.3879,B 24.9448,C -1.7165,E1 24.9028,E2 322.8016} C_DIS
LIN {X -71.8089,Y 97.9798,Z 128,A 121.7045,B 24.9444,C -1.7227,E1 24.9065,E2 324.4764} C_DIS
LIN {X -68.0928,Y 100.5979,Z 128,A 119.5936,B 24.944,C -1.7284,E1 24.9113,E2 326.5807} C_DIS
LIN {X -65.3903,Y 102.3755,Z 128,A 118.0688,B 24.9438,C -1.7314,E1 24.9149,E2 328.1033} C_DIS
LIN {X -62.1695,Y 104.3632,Z 128,A 115.5991,B 24.9455,C -1.7049,E1 24.921,E2 330.6436} C_DIS
LIN {X -57.9754,Y 106.7493,Z 128,A 114.036,B 24.9433,C -1.74,E1 24.9246,E2 332.1277} C_DIS
LIN {X -55.3859,Y 108.1156,Z 128,A 112.5737,B 24.9433,C -1.7388,E1 24.9283,E2 333.597} C_DIS
LIN {X -52.3646,Y 109.6111,Z 128,A 110.996,B 24.9431,C -1.7418,E1 24.9322,E2 335.1715} C_DIS
LIN {X -48.2988,Y 111.4623,Z 128,A 108.9092,B 24.9429,C -1.7459,E1 24.9375,E2 337.2536} C_DIS
LIN {X -44.4124,Y 113.0668,Z 128,A 107.194,B 24.9419,C -1.7606,E1 24.9419,E2 338.9377} C_DIS
LIN {X -41.7081,Y 114.0921,Z 128,A 105.5608,B 24.9426,C -1.7505,E1 24.9462,E2 340.5985} C_DIS
LIN {X -38.3248,Y 115.2737,Z 128,A 103.8826,B 24.9424,C -1.7531,E1 24.9506,E2 342.2736} C_DIS
LIN {X -34.9284,Y 116.3474,Z 128,A 102.1759,B 24.9424,C -1.7538,E1 24.9552,E2 343.9815} C_DIS
LIN {X -31.6152,Y 117.2904,Z 128,A 100.5238,B 24.9424,C -1.7544,E1 24.9596,E2 345.635} C_DIS
LIN {X -28.623,Y 118.0564,Z 128,A 99.1807,B 24.9419,C -1.7609,E1 24.9632,E2 346.9645} C_DIS
LIN {X -25.9268,Y 118.6776,Z 128,A 97.7223,B 24.9423,C -1.7552,E1 24.9673,E2 348.4382} C_DIS
LIN {X -22.662,Y 119.3444,Z 128,A 96.147,B 24.9422,C -1.7563,E1 24.9716,E2 350.0127} C_DIS
LIN {X -16.2664,Y 120.3844,Z 128,A 92.9603,B 24.9424,C -1.7525,E1 24.9804,E2 353.2112} C_DIS
LIN {X -9.3595,Y 121.1159,Z 128,A 90.0235,B 24.9413,C -1.7696,E1 24.9885,E2 356.1091} C_DIS
LIN {X -2.8047,Y 121.4455,Z 128,A 86.8101,B 24.9416,C -1.7652,E1 24.9975,E2 359.3336} C_DIS
LIN {X 2.8693,Y 121.4443,Z 128,A 84.0551,B 24.9418,C -1.762,E1 25.0052,E2 362.0959} C_DIS
LIN {X 8.8144,Y 121.158,Z 128,A 81.3404,B 24.9415,C -1.7663,E1 25.0127,E2 364.7994} C_DIS
LIN {X 15.2183,Y 120.5202,Z 128,A 78.4226,B 24.9412,C -1.7713,E1 25.0208,E2 367.7035} C_DIS
LIN {X 20.0677,Y 119.8075,Z 128,A 75.9223,B 24.9418,C -1.7619,E1 25.0277,E2 370.2237} C_DIS
LIN {X 23.5881,Y 119.1661,Z 128,A 74.0943,B 24.9423,C -1.7547,E1 25.0328,E2 372.0667} C_DIS
LIN {X 27.2895,Y 118.3716,Z 128,A 72.444,B 24.9419,C -1.76,E1 25.0372,E2 373.7021} C_DIS
LIN {X 30.8882,Y 117.4859,Z 128,A 70.596,B 24.9423,C -1.7543,E1 25.0423,E2 375.5609} C_DIS
LIN {X 35.0123,Y 116.3225,Z 128,A 68.7176,B 24.942,C -1.7595,E1 25.0473,E2 377.4239} C_DIS
LIN {X 37.7651,Y 115.4578,Z 128,A 67.36,B 24.942,C -1.7586,E1 25.0509,E2 378.7811} C_DIS
LIN {X 40.4372,Y 114.5489,Z 128,A 66.0249,B 24.9421,C -1.7572,E1 25.0544,E2 380.1168} C_DIS
LIN {X 43.879,Y 113.2763,Z 128,A 64.3874,B 24.942,C -1.7599,E1 25.0586,E2 381.7444} C_DIS
LIN {X 48.2112,Y 111.5005,Z 128,A 62.106,B 24.9423,C -1.7541,E1 25.0646,E2 384.0342} C_DIS
LIN {X 51.2685,Y 110.1276,Z 128,A 60.5095,B 24.9425,C -1.7515,E1 25.0686,E2 385.6328} C_DIS
LIN {X 54.2186,Y 108.706,Z 128,A 59.0238,B 24.9425,C -1.7523,E1 25.0723,E2 387.1127} C_DIS
LIN {X 56.5118,Y 107.5313,Z 128,A 57.7882,B 24.9426,C -1.7498,E1 25.0754,E2 388.3508} C_DIS
LIN {X 59.2352,Y 106.0554,Z 128,A 56.2848,B 24.9429,C -1.7457,E1 25.0791,E2 389.8595} C_DIS
LIN {X 62.5391,Y 104.1433,Z 128,A 54.3069,B 24.9436,C -1.7346,E1 25.0839,E2 391.8576} C_DIS
LIN {X 65.2664,Y 102.455,Z 128,A 52.057,B 24.946,C -1.6974,E1 25.0894,E2 394.1881} C_DIS
LIN {X 70.2749,Y 99.0864,Z 128,A 50.3558,B 24.9428,C -1.7469,E1 25.093,E2 395.7666} C_DIS
LIN {X 72.9221,Y 97.1541,Z 128,A 48.6201,B 24.9436,C -1.735,E1 25.0969,E2 397.5241} C_DIS
LIN {X 75.8463,Y 94.8912,Z 128,A 46.8717,B 24.9438,C -1.7315,E1 25.1008,E2 399.2743} C_DIS
LIN {X 78.6642,Y 92.5664,Z 128,A 45.1606,B 24.944,C -1.7288,E1 25.1045,E2 400.9853} C_DIS
LIN {X 81.2387,Y 90.3156,Z 128,A 43.557,B 24.9442,C -1.726,E1 25.1078,E2 402.5892} C_DIS
LIN {X 84.0207,Y 87.7339,Z 128,A 41.6753,B 24.9447,C -1.7178,E1 25.1117,E2 404.4824} C_DIS
LIN {X 86.337,Y 85.4546,Z 128,A 39.5459,B 24.9467,C -1.6858,E1 25.116,E2 406.6782} C_DIS
LIN {X 89.7676,Y 81.8443,Z 128,A 37.9742,B 24.9447,C -1.7179,E1 25.1188,E2 408.1673} C_DIS
LIN {X 91.6173,Y 79.7675,Z 128,A 36.5841,B 24.9451,C -1.7111,E1 25.1214,E2 409.5673} C_DIS
LIN {X 93.7314,Y 77.2736,Z 128,A 35.1245,B 24.9451,C -1.7114,E1 25.124,E2 411.0195} C_DIS
LIN {X 95.2838,Y 75.3496,Z 128,A 33.8509,B 24.9456,C -1.7033,E1 25.1262,E2 412.3061} C_DIS
LIN {X 97.2801,Y 72.7545,Z 128,A 32.409,B 24.9456,C -1.7045,E1 25.1286,E2 413.7385} C_DIS
LIN {X 98.948,Y 70.4689,Z 128,A 31.0018,B 24.946,C -1.6976,E1 25.1309,E2 415.1551} C_DIS
LIN {X 101.6872,Y 66.4568,Z 128,A 28.795,B 24.9461,C -1.6957,E1 25.1344,E2 417.3553} C_DIS
LIN {X 104.553,Y 61.8484,Z 128,A 25.7902,B 24.9479,C -1.6671,E1 25.1388,E2 420.4122} C_DIS
LIN {X 106.4444,Y 58.5374,Z 128,A 24.4841,B 24.9467,C -1.6862,E1 25.1405,E2 421.6666} C_DIS
LIN {X 107.7145,Y 56.1639,Z 128,A 23.075,B 24.9474,C -1.6758,E1 25.1424,E2 423.0927} C_DIS
LIN {X 109.477,Y 52.6435,Z 128,A 21.3085,B 24.9474,C -1.675,E1 25.1445,E2 424.8518} C_DIS
LIN {X 110.9376,Y 49.4936,Z 128,A 19.5802,B 24.948,C -1.6658,E1 25.1465,E2 426.5924} C_DIS
LIN {X 112.6331,Y 45.5022,Z 128,A 17.6613,B 24.948,C -1.666,E1 25.1486,E2 428.5003} C_DIS
LIN {X 114.1705,Y 41.4931,Z 128,A 15.6159,B 24.9484,C -1.6589,E1 25.1506,E2 430.5508} C_DIS
LIN {X 115.2436,Y 38.4142,Z 128,A 14.0464,B 24.9488,C -1.6527,E1 25.152,E2 432.1262} C_DIS
LIN {X 116.353,Y 34.9095,Z 128,A 12.3108,B 24.9492,C -1.6473,E1 25.1534,E2 433.8646} C_DIS
LIN {X 117.4254,Y 31.1155,Z 128,A 10.5842,B 24.9492,C -1.6481,E1 25.1547,E2 435.5794} C_DIS
LIN {X 118.2718,Y 27.7217,Z 128,A 8.8676,B 24.9496,C -1.6396,E1 25.1559,E2 437.306} C_DIS
LIN {X 119.0321,Y 24.2477,Z 128,A 7.2202,B 24.9499,C -1.6358,E1 25.1568,E2 438.9528} C_DIS
LIN {X 119.6417,Y 21.039,Z 128,A 5.7714,B 24.9499,C -1.6355,E1 25.1575,E2 440.394} C_DIS
LIN {X 120.1944,Y 17.611,Z 128,A 3.682,B 24.9516,C -1.6079,E1 25.1584,E2 442.5362} C_DIS
LIN {X 120.652,Y 14.1297,Z 128,A 2.2239,B 24.9513,C -1.6123,E1 25.1589,E2 443.9751} C_DIS
LIN {X 121.1074,Y 9.4663,Z 128,A 0.2444,B 24.951,C -1.6166,E1 25.1594,E2 445.9328} C_DIS
LIN {X 121.367,Y 5.1594,Z 128,A -1.7549,B 24.9513,C -1.6117,E1 25.1597,E2 447.9317} C_DIS
LIN {X 121.4786,Y 0.0706,Z 128,A -4.1095,B 24.9517,C -1.6062,E1 25.1597,E2 450.2855} C_DIS
LIN {X 121.3908,Y -4.5991,Z 128,A -6.2417,B 24.9519,C -1.6024,E1 25.1597,E2 452.4138} C_DIS
LIN {X 121.2557,Y -7.3497,Z 128,A -7.7453,B 24.9528,C -1.588,E1 25.1594,E2 453.9425} C_DIS
LIN {X 120.7705,Y -13.0855,Z 128,A -10.0818,B 24.9522,C -1.598,E1 25.1588,E2 456.2416} C_DIS
LIN {X 120.22,Y -17.4306,Z 128,A -12.4078,B 24.9533,C -1.5782,E1 25.158,E2 458.6004} C_DIS
LIN {X 119.1138,Y -23.8496,Z 128,A -15.3318,B 24.9535,C -1.5755,E1 25.1566,E2 461.5136} C_DIS
LIN {X 118.2724,Y -27.719,Z 128,A -17.2422,B 24.954,C -1.5674,E1 25.1554,E2 463.4322} C_DIS
LIN {X 117.4379,Y -31.0693,Z 128,A -19.0632,B 24.9548,C -1.5525,E1 25.1541,E2 465.2777} C_DIS
LIN {X 116.2985,Y -35.0933,Z 128,A -20.7945,B 24.9545,C -1.5582,E1 25.1528,E2 466.9857} C_DIS
LIN {X 115.5454,Y -37.4942,Z 128,A -22.0893,B 24.955,C -1.5491,E1 25.1517,E2 468.2946} C_DIS
LIN {X 114.4496,Y -40.72,Z 128,A -23.6162,B 24.9551,C -1.5479,E1 25.1503,E2 469.8157} C_DIS
LIN {X 112.985,Y -44.6206,Z 128,A -25.4893,B 24.9551,C -1.5464,E1 25.1484,E2 471.6821} C_DIS
LIN {X 110.0339,Y -51.47,Z 128,A -28.9937,B 24.9558,C -1.5361,E1 25.1445,E2 475.1915} C_DIS
LIN {X 108.8079,Y -54.013,Z 128,A -30.4069,B 24.9563,C -1.528,E1 25.1427,E2 476.6162} C_DIS
LIN {X 107.2894,Y -56.9711,Z 128,A -32.0536,B 24.9568,C -1.5194,E1 25.1406,E2 478.2746} C_DIS
LIN {X 105.5428,Y -60.1454,Z 128,A -33.5311,B 24.9564,C -1.5258,E1 25.1386,E2 479.7292} C_DIS
LIN {X 104.1122,Y -62.5903,Z 128,A -35.0302,B 24.9571,C -1.5138,E1 25.1364,E2 481.249} C_DIS
LIN {X 101.9789,Y -66.0082,Z 128,A -37.0046,B 24.9576,C -1.5046,E1 25.1335,E2 483.235} C_DIS
LIN {X 99.6165,Y -69.521,Z 128,A -39.5227,B 24.9593,C -1.4734,E1 25.1294,E2 485.8144} C_DIS
LIN {X 96.7785,Y -73.4221,Z 128,A -41.0646,B 24.9577,C -1.5031,E1 25.1269,E2 487.2788} C_DIS
LIN {X 95.2107,Y -75.442,Z 128,A -42.29,B 24.9579,C -1.4989,E1 25.1248,E2 488.5083} C_DIS
LIN {X 93.354,Y -77.7277,Z 128,A -43.6841,B 24.9581,C -1.4949,E1 25.1223,E2 489.9054} C_DIS
LIN {X 90.9975,Y -80.4768,Z 128,A -45.75,B 24.9594,C -1.4728,E1 25.1185,E2 492.0141} C_DIS
LIN {X 88.8425,Y -82.8483,Z 128,A -47.1165,B 24.9592,C -1.4761,E1 25.1159,E2 493.367} C_DIS
LIN {X 85.3907,Y -86.4001,Z 128,A -49.227,B 24.9589,C -1.4814,E1 25.1118,E2 495.4561} C_DIS
LIN {X 82.8424,Y -88.848,Z 128,A -50.9892,B 24.9594,C -1.4726,E1 25.1082,E2 497.2316} C_DIS
LIN {X 79.3745,Y -91.9599,Z 128,A -53.3311,B 24.96,C -1.4604,E1 25.1032,E2 499.593} C_DIS
LIN {X 76.3532,Y -94.4816,Z 128,A -54.9689,B 24.9597,C -1.4669,E1 25.0997,E2 501.2093} C_DIS
LIN {X 72.9424,Y -97.1389,Z 128,A -56.9418,B 24.9597,C -1.4657,E1 25.0954,E2 503.1778} C_DIS
LIN {X 67.8183,Y -100.7837,Z 128,A -59.8941,B 24.9601,C -1.4602,E1 25.0886,E2 506.1328} C_DIS
LIN {X 64.5207,Y -102.9256,Z 128,A -61.7844,B 24.9603,C -1.4549,E1 25.0842,E2 508.0296} C_DIS
LIN {X 61.5158,Y -104.7496,Z 128,A -63.3562,B 24.9603,C -1.4559,E1 25.0804,E2 509.5941} C_DIS
LIN {X 58.5109,Y -106.4588,Z 128,A -65.2494,B 24.9611,C -1.4403,E1 25.0757,E2 511.5188} C_DIS
LIN {X 54.9091,Y -108.3592,Z 128,A -66.8971,B 24.9606,C -1.4502,E1 25.0717,E2 513.1384} C_DIS
LIN {X 52.2593,Y -109.6616,Z 128,A -68.4564,B 24.9612,C -1.4399,E1 25.0677,E2 514.718} C_DIS
LIN {X 46.5054,Y -112.2245,Z 128,A -71.2733,B 24.961,C -1.4427,E1 25.0606,E2 517.5213} C_DIS
LIN {X 43.1075,Y -113.5707,Z 128,A -73.094,B 24.9614,C -1.4357,E1 25.0558,E2 519.3547} C_DIS
LIN {X 35.492,Y -116.1772,Z 128,A -76.5579,B 24.9608,C -1.4468,E1 25.0467,E2 522.7856} C_DIS
LIN {X 31.1139,Y -117.4258,Z 128,A -79.0791,B 24.9619,C -1.4266,E1 25.0398,E2 525.3505} C_DIS
LIN {X 26.8527,Y -118.4725,Z 128,A -80.944,B 24.9615,C -1.4343,E1 25.0348,E2 527.1945} C_DIS
LIN {X 23.6993,Y -119.1447,Z 128,A -83.0116,B 24.9629,C -1.407,E1 25.029,E2 529.3241} C_DIS
LIN {X 19.9588,Y -119.8257,Z 128,A -84.3279,B 24.9618,C -1.4282,E1 25.0255,E2 530.589} C_DIS
LIN {X 16.2539,Y -120.386,Z 128,A -86.0571,B 24.9618,C -1.4287,E1 25.0207,E2 532.3153} C_DIS
LIN {X 13.5415,Y -120.7209,Z 128,A -87.3153,B 24.9618,C -1.4294,E1 25.0172,E2 533.5711} C_DIS
LIN {X 10.8694,Y -120.9897,Z 128,A -88.7347,B 24.9621,C -1.4215,E1 25.0132,E2 535.0082} C_DIS
LIN {X 6.1318,Y -121.3231,Z 128,A -90.7917,B 24.9617,C -1.4291,E1 25.0076,E2 537.0464} C_DIS
LIN {X 3.3194,Y -121.4319,Z 128,A -92.4587,B 24.9626,C -1.4128,E1 25.0028,E2 538.7516} C_DIS
LIN {X 3.3194,Y -121.4319,Z 128,A -92.4587,B 24.9626,C -1.4128,E1 25.0028,E2 538.7516} C_DIS
Enddeposition()
LIN {X 0.8378,Y -120.6067,Z 128,A -92.2955,B 24.9584,C -1.4903,E1 25.0038,E2 538.4048} C_DIS
Startdeposition()
$VEL.CP = VEL_PRINT
LIN {X 5.1981,Y -120.5129,Z 128,A -90.7796,B 24.9598,C -1.4645,E1 25.0078,E2 536.9504} C_DIS
LIN {X 11.7883,Y -120.0496,Z 128,A -87.3419,B 24.959,C -1.4801,E1 25.0175,E2 533.4776} C_DIS
LIN {X 15.3533,Y -119.644,Z 128,A -85.5098,B 24.9586,C -1.4873,E1 25.0226,E2 531.6298} C_DIS
LIN {X 20.1941,Y -118.923,Z 128,A -83.1206,B 24.9583,C -1.4921,E1 25.0292,E2 529.2315} C_DIS
LIN {X 23.5332,Y -118.3094,Z 128,A -81.6849,B 24.9587,C -1.485,E1 25.0331,E2 527.8145} C_DIS
LIN {X 27.3208,Y -117.4904,Z 128,A -80.0135,B 24.959,C -1.4786,E1 25.0376,E2 526.1603} C_DIS
LIN {X 31.1547,Y -116.5327,Z 128,A -78.1986,B 24.959,C -1.4776,E1 25.0425,E2 524.3506} C_DIS
LIN {X 34.2456,Y -115.6617,Z 128,A -76.7121,B 24.9591,C -1.4775,E1 25.0465,E2 522.8669} C_DIS
LIN {X 42.2687,Y -112.9777,Z 128,A -72.4347,B 24.9581,C -1.495,E1 25.0579,E2 518.5565} C_DIS
LIN {X 45.7305,Y -111.6207,Z 128,A -70.9537,B 24.9588,C -1.4837,E1 25.0616,E2 517.1055} C_DIS
LIN {X 50.7674,Y -109.4216,Z 128,A -68.2126,B 24.9582,C -1.494,E1 25.0687,E2 514.3468} C_DIS
LIN {X 54.192,Y -107.7687,Z 128,A -66.3164,B 24.9578,C -1.5014,E1 25.0734,E2 512.4384} C_DIS
LIN {X 59.3724,Y -105.0034,Z 128,A -63.5909,B 24.9577,C -1.5032,E1 25.0801,E2 509.7164} C_DIS
LIN {X 62.6888,Y -103.0558,Z 128,A -61.3838,B 24.9564,C -1.5253,E1 25.0855,E2 507.4639} C_DIS
LIN {X 65.9981,Y -100.9696,Z 128,A -59.956,B 24.9574,C -1.5078,E1 25.0887,E2 506.0821} C_DIS
LIN {X 70.2524,Y -98.0563,Z 128,A -56.5988,B 24.9545,C -1.5578,E1 25.0966,E2 502.6185} C_DIS
LIN {X 75.2188,Y -94.3017,Z 128,A -54.6496,B 24.957,C -1.5143,E1 25.1007,E2 500.7792} C_DIS
LIN {X 77.812,Y -92.1728,Z 128,A -52.6456,B 24.9557,C -1.5382,E1 25.1051,E2 498.7265} C_DIS
LIN {X 80.401,Y -89.9226,Z 128,A -51.7048,B 24.9574,C -1.5081,E1 25.1069,E2 497.8606} C_DIS
LIN {X 83.882,Y -86.6847,Z 128,A -49.1106,B 24.9561,C -1.53,E1 25.1123,E2 495.2252} C_DIS
LIN {X 85.6757,Y -84.9123,Z 128,A -47.1779,B 24.9538,C -1.5696,E1 25.1162,E2 493.2074} C_DIS
LIN {X 89.4369,Y -80.9435,Z 128,A -45.1818,B 24.9552,C -1.5462,E1 25.1198,E2 491.2754} C_DIS
LIN {X 93.5408,Y -76.1615,Z 128,A -42.649,B 24.9561,C -1.5313,E1 25.1243,E2 488.7892} C_DIS
LIN {X 96.4161,Y -72.4867,Z 128,A -39.7902,B 24.9539,C -1.5693,E1 25.1293,E2 485.8544} C_DIS
LIN {X 98.6333,Y -69.4433,Z 128,A -38.4145,B 24.9548,C -1.5537,E1 25.1315,E2 484.5223} C_DIS
LIN {X 101.0608,Y -65.8598,Z 128,A -36.4411,B 24.9547,C -1.5554,E1 25.1345,E2 482.5545} C_DIS
LIN {X 103.4617,Y -62.021,Z 128,A -34.1592,B 24.9539,C -1.5682,E1 25.1379,E2 480.2541} C_DIS
LIN {X 105.9088,Y -57.7389,Z 128,A -31.9133,B 24.9538,C -1.5703,E1 25.1409,E2 478.0148} C_DIS
LIN {X 107.2889,Y -55.1321,Z 128,A -30.4622,B 24.9534,C -1.577,E1 25.1428,E2 476.5555} C_DIS
LIN {X 109.4823,Y -50.6369,Z 128,A -27.7335,B 24.9519,C -1.602,E1 25.1461,E2 473.7828} C_DIS
LIN {X 110.9961,Y -47.2273,Z 128,A -26.2738,B 24.9525,C -1.5918,E1 25.1477,E2 472.3551} C_DIS
LIN {X 112.6886,Y -43.0322,Z 128,A -24.4555,B 24.9531,C -1.582,E1 25.1495,E2 470.57} C_DIS
LIN {X 113.7295,Y -40.2001,Z 128,A -22.8299,B 24.9523,C -1.5961,E1 25.1511,E2 468.9202} C_DIS
LIN {X 114.8302,Y -36.9385,Z 128,A -21.1978,B 24.952,C -1.6012,E1 25.1525,E2 467.2853} C_DIS
LIN {X 116.0076,Y -33.0554,Z 128,A -19.3007,B 24.9517,C -1.6058,E1 25.154,E2 465.3882} C_DIS
LIN {X 116.8571,Y -29.9133,Z 128,A -17.7397,B 24.9513,C -1.6116,E1 25.1551,E2 463.8226} C_DIS
LIN {X 117.7585,Y -26.1441,Z 128,A -15.9049,B 24.951,C -1.6172,E1 25.1563,E2 461.9852} C_DIS
LIN {X 118.4466,Y -22.8207,Z 128,A -14.239,B 24.9505,C -1.6252,E1 25.1572,E2 460.3102} C_DIS
LIN {X 119.6051,Y -15.6534,Z 128,A -10.8123,B 24.9499,C -1.6353,E1 25.1586,E2 456.8798} C_DIS
LIN {X 120.4144,Y -7.1403,Z 128,A -5.944,B 24.9465,C -1.6893,E1 25.1597,E2 451.9131} C_DIS
LIN {X 120.6209,Y -1.0581,Z 128,A -4.2042,B 24.9496,C -1.6408,E1 25.1597,E2 450.298} C_DIS
LIN {X 120.5099,Y 5.2678,Z 128,A -1.0907,B 24.9486,C -1.6559,E1 25.1597,E2 447.1674} C_DIS
LIN {X 120.3594,Y 8.001,Z 128,A 0.5506,B 24.9473,C -1.6772,E1 25.1593,E2 445.4855} C_DIS
LIN {X 120.085,Y 11.4046,Z 128,A 2.731,B 24.9452,C -1.7107,E1 25.1587,E2 443.2392} C_DIS
LIN {X 119.4126,Y 17.059,Z 128,A 4.5989,B 24.9473,C -1.6772,E1 25.158,E2 441.4612} C_DIS
LIN {X 118.7655,Y 21.0997,Z 128,A 6.5459,B 24.9469,C -1.6836,E1 25.1571,E2 439.5106} C_DIS
LIN {X 118.019,Y 24.948,Z 128,A 8.4549,B 24.9464,C -1.6918,E1 25.156,E2 437.5935} C_DIS
LIN {X 117.1809,Y 28.6186,Z 128,A 10.1589,B 24.9463,C -1.6932,E1 25.1549,E2 435.896} C_DIS
LIN {X 116.1707,Y 32.4796,Z 128,A 11.9406,B 24.9463,C -1.6934,E1 25.1536,E2 434.124} C_DIS
LIN {X 115.2034,Y 35.7569,Z 128,A 13.6386,B 24.9457,C -1.7021,E1 25.1523,E2 432.4152} C_DIS
LIN {X 114.0326,Y 39.3363,Z 128,A 15.3818,B 24.9455,C -1.7053,E1 25.1507,E2 430.6744} C_DIS
LIN {X 111.8725,Y 45.1119,Z 128,A 18.7851,B 24.9434,C -1.7376,E1 25.1472,E2 427.2138} C_DIS
LIN {X 110.3076,Y 48.8166,Z 128,A 20.3155,B 24.9443,C -1.7242,E1 25.1456,E2 425.7232} C_DIS
LIN {X 108.7838,Y 52.1199,Z 128,A 21.9197,B 24.9443,C -1.7231,E1 25.1437,E2 424.1303} C_DIS
LIN {X 107.2642,Y 55.1804,Z 128,A 23.63,B 24.9438,C -1.732,E1 25.1415,E2 422.4082} C_DIS
LIN {X 105.7188,Y 58.0891,Z 128,A 25.6241,B 24.9421,C -1.7576,E1 25.1388,E2 420.3641} C_DIS
LIN {X 103.6676,Y 61.6727,Z 128,A 27.3033,B 24.9427,C -1.7489,E1 25.1364,E2 418.7139} C_DIS
LIN {X 100.9912,Y 65.9654,Z 128,A 29.4504,B 24.9431,C -1.7427,E1 25.1332,E2 416.5924} C_DIS
LIN {X 98.8126,Y 69.1853,Z 128,A 31.2326,B 24.943,C -1.7443,E1 25.1304,E2 414.8152} C_DIS
LIN {X 96.7693,Y 72.0164,Z 128,A 32.9852,B 24.9424,C -1.753,E1 25.1275,E2 413.0503} C_DIS
LIN {X 94.6567,Y 74.7696,Z 128,A 34.4577,B 24.9427,C -1.7485,E1 25.125,E2 411.5955} C_DIS
LIN {X 92.117,Y 77.8785,Z 128,A 36.4736,B 24.9421,C -1.7584,E1 25.1214,E2 409.5656} C_DIS
LIN {X 89.9166,Y 80.4077,Z 128,A 38.0018,B 24.9421,C -1.7589,E1 25.1186,E2 408.0429} C_DIS
LIN {X 87.1522,Y 83.397,Z 128,A 40.1418,B 24.9411,C -1.7733,E1 25.1144,E2 405.8784} C_DIS
LIN {X 83.6537,Y 86.9048,Z 128,A 42.2931,B 24.9414,C -1.7686,E1 25.1102,E2 403.7473} C_DIS
LIN {X 80.9347,Y 89.4448,Z 128,A 44.1612,B 24.9408,C -1.7771,E1 25.1063,E2 401.8667} C_DIS
LIN {X 78.3477,Y 91.7172,Z 128,A 45.6818,B 24.941,C -1.7748,E1 25.1031,E2 400.3574} C_DIS
LIN {X 75.9931,Y 93.6772,Z 128,A 47.1841,B 24.9406,C -1.7798,E1 25.0999,E2 398.8489} C_DIS
LIN {X 72.9124,Y 96.0963,Z 128,A 49.0728,B 24.9403,C -1.7846,E1 25.0957,E2 396.9559} C_DIS
LIN {X 70.1109,Y 98.1573,Z 128,A 51.2888,B 24.9383,C -1.8148,E1 25.0905,E2 394.6763} C_DIS
LIN {X 66.1997,Y 100.8367,Z 128,A 53.0137,B 24.9397,C -1.793,E1 25.0866,E2 393.0086} C_DIS
LIN {X 62.9061,Y 102.9237,Z 128,A 54.8533,B 24.9396,C -1.7953,E1 25.0822,E2 391.1695} C_DIS
LIN {X 59.1269,Y 105.1405,Z 128,A 56.8044,B 24.9398,C -1.7921,E1 25.0776,E2 389.2318} C_DIS
LIN {X 56.1255,Y 106.7723,Z 128,A 58.4321,B 24.9396,C -1.7945,E1 25.0735,E2 387.6029} C_DIS
LIN {X 52.5636,Y 108.5706,Z 128,A 60.288,B 24.9396,C -1.7951,E1 25.0689,E2 385.7507} C_DIS
LIN {X 49.6102,Y 109.951,Z 128,A 61.8654,B 24.9394,C -1.7983,E1 25.0649,E2 384.1697} C_DIS
LIN {X 47.2836,Y 110.9724,Z 128,A 63.4811,B 24.938,C -1.819,E1 25.0606,E2 382.5088} C_DIS
LIN {X 43.9578,Y 112.3304,Z 128,A 64.9777,B 24.9385,C -1.8108,E1 25.0568,E2 381.035} C_DIS
LIN {X 39.9456,Y 113.8188,Z 128,A 66.8162,B 24.939,C -1.8035,E1 25.052,E2 379.2176} C_DIS
LIN {X 36.0317,Y 115.1182,Z 128,A 68.5266,B 24.9397,C -1.7934,E1 25.0476,E2 377.5342} C_DIS
LIN {X 32.1817,Y 116.2551,Z 128,A 70.7987,B 24.9385,C -1.8118,E1 25.0414,E2 375.2224} C_DIS
LIN {X 28.5766,Y 117.1911,Z 128,A 72.3813,B 24.939,C -1.8042,E1 25.0371,E2 373.6602} C_DIS
LIN {X 25.4866,Y 117.9019,Z 128,A 73.941,B 24.9388,C -1.8075,E1 25.0329,E2 372.0947} C_DIS
LIN {X 21.6086,Y 118.674,Z 128,A 75.816,B 24.9388,C -1.8081,E1 25.0277,E2 370.2205} C_DIS
LIN {X 18.8485,Y 119.144,Z 128,A 77.1924,B 24.9385,C -1.8107,E1 25.0239,E2 368.8393} C_DIS
LIN {X 14.7109,Y 119.7265,Z 128,A 79.911,B 24.9362,C -1.8454,E1 25.0162,E2 366.0406} C_DIS
LIN {X 9.4034,Y 120.2581,Z 128,A 81.6222,B 24.9388,C -1.8073,E1 25.0116,E2 364.4206} C_DIS
LIN {X 3.3806,Y 120.578,Z 128,A 84.2976,B 24.9394,C -1.7985,E1 25.0043,E2 361.767} C_DIS
LIN {X -2.5465,Y 120.5985,Z 128,A 87.2846,B 24.9389,C -1.8057,E1 24.9959,E2 358.763} C_DIS
LIN {X -9.6547,Y 120.238,Z 128,A 90.3332,B 24.94,C -1.7892,E1 24.9875,E2 355.7526} C_DIS
LIN {X -15.4028,Y 119.6376,Z 128,A 93.4086,B 24.9391,C -1.8026,E1 24.9788,E2 352.6436} C_DIS
LIN {X -18.7071,Y 119.1658,Z 128,A 95.203,B 24.9385,C -1.811,E1 24.9738,E2 350.8277} C_DIS
LIN {X -22.5844,Y 118.4921,Z 128,A 96.9653,B 24.939,C -1.8047,E1 24.969,E2 349.0786} C_DIS
LIN {X -26.4249,Y 117.6973,Z 128,A 98.9351,B 24.9387,C -1.8079,E1 24.9636,E2 347.0989} C_DIS
LIN {X -29.4537,Y 116.9753,Z 128,A 100.4033,B 24.9389,C -1.8059,E1 24.9596,E2 345.6332} C_DIS
LIN {X -33.3364,Y 115.9279,Z 128,A 102.275,B 24.9391,C -1.8022,E1 24.9546,E2 343.7674} C_DIS
LIN {X -36.7326,Y 114.8968,Z 128,A 103.9062,B 24.9394,C -1.7978,E1 24.9503,E2 342.1439} C_DIS
LIN {X -39.7908,Y 113.8732,Z 128,A 105.4837,B 24.9394,C -1.7979,E1 24.9461,E2 340.563} C_DIS
LIN {X -42.3931,Y 112.9306,Z 128,A 107.2307,B 24.9382,C -1.8155,E1 24.9414,E2 338.7704} C_DIS
LIN {X -46.2099,Y 111.4248,Z 128,A 108.7984,B 24.9396,C -1.7956,E1 24.9375,E2 337.2465} C_DIS
LIN {X -49.321,Y 110.0813,Z 128,A 110.6697,B 24.9389,C -1.8049,E1 24.9327,E2 335.3486} C_DIS
LIN {X -52.4013,Y 108.6486,Z 128,A 111.9221,B 24.9402,C -1.7863,E1 24.9296,E2 334.1374} C_DIS
LIN {X -55.7719,Y 106.9585,Z 128,A 113.7728,B 24.9402,C -1.7859,E1 24.925,E2 332.2824} C_DIS
LIN {X -60.0614,Y 104.6089,Z 128,A 116.2361,B 24.9401,C -1.788,E1 24.919,E2 329.807} C_DIS
LIN {X -63.8572,Y 102.3359,Z 128,A 118.2143,B 24.9407,C -1.7787,E1 24.9143,E2 327.845} C_DIS
LIN {X -67.3156,Y 100.0956,Z 128,A 119.9246,B 24.9417,C -1.764,E1 24.9104,E2 326.164} C_DIS
LIN {X -71.1207,Y 97.4282,Z 128,A 122.3115,B 24.9415,C -1.7673,E1 24.9049,E2 323.761} C_DIS
LIN {X -73.5479,Y 95.6091,Z 128,A 124.1924,B 24.9404,C -1.7836,E1 24.9006,E2 321.8346} C_DIS
LIN {X -76.4139,Y 93.3362,Z 128,A 125.6534,B 24.9414,C -1.7675,E1 24.8975,E2 320.4062} C_DIS
LIN {X -79.9059,Y 90.3656,Z 128,A 127.722,B 24.9421,C -1.7578,E1 24.8932,E2 318.3527} C_DIS
LIN {X -82.2443,Y 88.2414,Z 128,A 129.2988,B 24.9421,C -1.7576,E1 24.8899,E2 316.77} C_DIS
LIN {X -86.3609,Y 84.218,Z 128,A 132.0574,B 24.9425,C -1.7519,E1 24.8845,E2 314.0132} C_DIS
LIN {X -89.2917,Y 81.1033,Z 128,A 134.0979,B 24.9428,C -1.7472,E1 24.8806,E2 311.975} C_DIS
LIN {X -91.5406,Y 78.555,Z 128,A 135.9736,B 24.9423,C -1.7544,E1 24.8772,E2 310.0737} C_DIS
LIN {X -95.1926,Y 74.0884,Z 128,A 139.0238,B 24.9419,C -1.7605,E1 24.8718,E2 306.9945} C_DIS
LIN {X -97.9174,Y 70.447,Z 128,A 140.4166,B 24.9445,C -1.7212,E1 24.8697,E2 305.6886} C_DIS
LIN {X -100.2226,Y 67.128,Z 128,A 142.5971,B 24.9441,C -1.7271,E1 24.8662,E2 303.4833} C_DIS
LIN {X -102.2074,Y 64.063,Z 128,A 144.3504,B 24.9444,C -1.7229,E1 24.8636,E2 301.731} C_DIS
LIN {X -104.4858,Y 60.2755,Z 128,A 147.3544,B 24.9422,C -1.7561,E1 24.8593,E2 298.6322} C_DIS
LIN {X -107.4814,Y 54.7555,Z 128,A 148.9363,B 24.9467,C -1.6866,E1 24.8574,E2 297.2077} C_DIS
LIN {X -110.1482,Y 49.1725,Z 128,A 152.4476,B 24.9457,C -1.702,E1 24.8532,E2 293.6404} C_DIS
LIN {X -111.6493,Y 45.6601,Z 128,A 154.1138,B 24.9465,C -1.6901,E1 24.8514,E2 291.9935} C_DIS
LIN {X -114.7435,Y 37.2064,Z 128,A 158.4596,B 24.9471,C -1.6795,E1 24.8473,E2 287.6483} C_DIS
LIN {X -115.6275,Y 34.3609,Z 128,A 160.6403,B 24.9453,C -1.708,E1 24.8455,E2 285.387} C_DIS
LIN {X -117.0243,Y 29.2602,Z 128,A 162.4714,B 24.9477,C -1.6705,E1 24.8443,E2 283.6347} C_DIS
LIN {X -117.834,Y 25.7982,Z 128,A 164.0621,B 24.9483,C -1.6609,E1 24.8433,E2 282.0576} C_DIS
LIN {X -118.4682,Y 22.7085,Z 128,A 165.6223,B 24.9484,C -1.6587,E1 24.8424,E2 280.4935} C_DIS
LIN {X -119.1264,Y 18.9621,Z 128,A 167.4961,B 24.9486,C -1.6556,E1 24.8416,E2 278.6157} C_DIS
LIN {X -119.6149,Y 15.5775,Z 128,A 169.008,B 24.9493,C -1.6455,E1 24.841,E2 277.1189} C_DIS
LIN {X -119.9804,Y 12.4534,Z 128,A 170.6145,B 24.9493,C -1.6455,E1 24.8405,E2 275.5029} C_DIS
LIN {X -120.3337,Y 8.381,Z 128,A 172.5504,B 24.9497,C -1.6389,E1 24.8401,E2 273.5711} C_DIS
LIN {X -120.5215,Y 4.9992,Z 128,A 174.1794,B 24.9499,C -1.6345,E1 24.8399,E2 271.9428} C_DIS
LIN {X -120.6221,Y 0.8587,Z 128,A 176.0851,B 24.9505,C -1.6254,E1 24.8398,E2 270.0473} C_DIS
LIN {X -120.6044,Y -2.2272,Z 128,A 177.6064,B 24.9506,C -1.623,E1 24.8398,E2 268.5225} C_DIS
LIN {X -120.479,Y -5.9713,Z 128,A 179.5118,B 24.9506,C -1.6226,E1 24.8401,E2 266.6066} C_DIS
LIN {X -120.2481,Y -9.5276,Z 128,A -178.9813,B 24.9515,C -1.6091,E1 24.8404,E2 265.1227} C_DIS
LIN {X -119.9934,Y -12.3295,Z 128,A -177.519,B 24.9515,C -1.6102,E1 24.8408,E2 263.649} C_DIS
LIN {X -119.6087,Y -15.6253,Z 128,A -175.968,B 24.9518,C -1.6041,E1 24.8413,E2 262.1034} C_DIS
LIN {X -119.0287,Y -19.5617,Z 128,A -174.2717,B 24.9526,C -1.5897,E1 24.842,E2 260.4313} C_DIS
LIN {X -118.5796,Y -22.1284,Z 128,A -172.7151,B 24.9521,C -1.5995,E1 24.8428,E2 258.8422} C_DIS
LIN {X -117.884,Y -25.5689,Z 128,A -171.151,B 24.9526,C -1.5898,E1 24.8437,E2 257.2919} C_DIS
LIN {X -117.2584,Y -28.3007,Z 128,A -169.6433,B 24.9524,C -1.5932,E1 24.8447,E2 255.7672} C_DIS
LIN {X -114.9946,Y -36.4302,Z 128,A -165.6516,B 24.9532,C -1.5801,E1 24.8478,E2 251.7837} C_DIS
LIN {X -112.8184,Y -42.6894,Z 128,A -162.6334,B 24.9541,C -1.565,E1 24.8506,E2 248.7844} C_DIS
LIN {X -111.7227,Y -45.48,Z 128,A -161.148,B 24.9541,C -1.5635,E1 24.8521,E2 247.2943} C_DIS
LIN {X -110.3357,Y -48.7522,Z 128,A -159.2949,B 24.9541,C -1.5657,E1 24.8542,E2 245.4257} C_DIS
LIN {X -108.7827,Y -52.1223,Z 128,A -157.682,B 24.9547,C -1.5542,E1 24.8561,E2 243.8314} C_DIS
LIN {X -107.3181,Y -55.0749,Z 128,A -156.1236,B 24.955,C -1.5495,E1 24.8581,E2 242.2759} C_DIS
LIN {X -105.55,Y -58.3936,Z 128,A -154.4639,B 24.9556,C -1.539,E1 24.8602,E2 240.6324} C_DIS
LIN {X -103.5091,Y -61.941,Z 128,A -152.2363,B 24.9552,C -1.5461,E1 24.8634,E2 238.3763} C_DIS
LIN {X -101.5711,Y -65.0669,Z 128,A -150.2116,B 24.9548,C -1.5537,E1 24.8665,E2 236.3233} C_DIS
LIN {X -99.6302,Y -68.003,Z 128,A -148.8711,B 24.9559,C -1.5348,E1 24.8685,E2 235.0211} C_DIS
LIN {X -97.5519,Y -70.9518,Z 128,A -147.3883,B 24.9567,C -1.5204,E1 24.8709,E2 233.5654} C_DIS
LIN {X -94.8196,Y -74.5635,Z 128,A -144.9903,B 24.9564,C -1.5259,E1 24.875,E2 231.1429} C_DIS
LIN {X -92.6266,Y -77.2706,Z 128,A -143.4538,B 24.9569,C -1.5167,E1 24.8777,E2 229.6211} C_DIS
LIN {X -90.6208,Y -79.6139,Z 128,A -141.8141,B 24.9567,C -1.521,E1 24.8807,E2 227.9637} C_DIS
LIN {X -88.4645,Y -82.0048,Z 128,A -140.2217,B 24.9567,C -1.5204,E1 24.8838,E2 226.3659} C_DIS
LIN {X -85.8329,Y -84.7532,Z 128,A -138.5483,B 24.9573,C -1.5105,E1 24.887,E2 224.7087} C_DIS
LIN {X -83.4097,Y -87.14,Z 128,A -136.7783,B 24.9571,C -1.5139,E1 24.8906,E2 222.9232} C_DIS
LIN {X -80.5392,Y -89.7988,Z 128,A -135.0514,B 24.9576,C -1.5043,E1 24.8941,E2 221.2123} C_DIS
LIN {X -77.1446,Y -92.7313,Z 128,A -132.9128,B 24.9578,C -1.5005,E1 24.8986,E2 219.0744} C_DIS
LIN {X -74.1698,Y -95.1299,Z 128,A -131.0954,B 24.958,C -1.4972,E1 24.9026,E2 217.2581} C_DIS
LIN {X -71.4328,Y -97.1997,Z 128,A -129.4869,B 24.9582,C -1.4934,E1 24.9062,E2 215.6529} C_DIS
LIN {X -67.7941,Y -99.7716,Z 128,A -127.3652,B 24.9584,C -1.49,E1 24.9111,E2 213.532} C_DIS
LIN {X -65.3768,Y -101.3722,Z 128,A -126.0203,B 24.9586,C -1.4864,E1 24.9142,E2 212.1914} C_DIS
LIN {X -62.9969,Y -102.8686,Z 128,A -124.5631,B 24.9584,C -1.4898,E1 24.9177,E2 210.7214} C_DIS
LIN {X -59.937,Y -104.6803,Z 128,A -122.8806,B 24.9586,C -1.4871,E1 24.9218,E2 209.0404} C_DIS
LIN {X -56.3222,Y -106.6687,Z 128,A -120.905,B 24.9586,C -1.4852,E1 24.9266,E2 207.0637} C_DIS
LIN {X -52.8318,Y -108.4417,Z 128,A -118.9538,B 24.9586,C -1.487,E1 24.9315,E2 205.1031} C_DIS
LIN {X -49.9927,Y -109.7786,Z 128,A -117.1576,B 24.9579,C -1.4993,E1 24.9362,E2 203.2733} C_DIS
LIN {X -46.6595,Y -111.2354,Z 128,A -115.6015,B 24.9584,C -1.4896,E1 24.9401,E2 201.7367} C_DIS
LIN {X -42.2747,Y -112.9755,Z 128,A -113.5847,B 24.9591,C -1.4771,E1 24.9453,E2 199.7451} C_DIS
LIN {X -38.4245,Y -114.3414,Z 128,A -111.2692,B 24.9583,C -1.4928,E1 24.9515,E2 197.3881} C_DIS
LIN {X -34.9447,Y -115.4543,Z 128,A -109.799,B 24.959,C -1.4792,E1 24.9554,E2 195.9475} C_DIS
LIN {X -31.2974,Y -116.4941,Z 128,A -108.1023,B 24.9593,C -1.4733,E1 24.9599,E2 194.2624} C_DIS
LIN {X -27.4849,Y -117.4524,Z 128,A -106.239,B 24.9594,C -1.472,E1 24.965,E2 192.3994} C_DIS
LIN {X -24.4309,Y -118.1251,Z 128,A -104.7689,B 24.9594,C -1.4707,E1 24.969,E2 190.9308} C_DIS
LIN {X -20.0112,Y -118.9536,Z 128,A -102.5326,B 24.9593,C -1.4746,E1 24.9752,E2 188.6829} C_DIS
LIN {X -13.2377,Y -119.8983,Z 128,A -99.4478,B 24.9597,C -1.4662,E1 24.9837,E2 185.6156} C_DIS
LIN {X -7.0619,Y -120.4187,Z 128,A -96.6219,B 24.96,C -1.4606,E1 24.9915,E2 182.8018} C_DIS
LIN {X -1.7115,Y -120.6139,Z 128,A -93.9272,B 24.9596,C -1.468,E1 24.9991,E2 180.0891} C_DIS
LIN {X 0.8378,Y -120.6067,Z 128,A -92.2915,B 24.9585,C -1.4886,E1 25.0038,E2 178.4048} C_DIS
Enddeposition()
LIN {X 0.8378,Y -120.6067,Z 128,A -92.2915,B 24.9585,C -1.4886,E1 25.0038,E2 178.4048} C_DIS
Startdeposition()
$VEL.CP = VEL_PRINT
LIN {X -0.2135,Y -119.7743,Z 128,A -94.7106,B 24.9625,C -1.4143,E1 24.9966,E2 180.9998} C_DIS
LIN {X -5.4463,Y -119.6498,Z 128,A -96.284,B 24.9603,C -1.4565,E1 24.9924,E2 182.4737} C_DIS
LIN {X -10.3367,Y -119.3284,Z 128,A -98.9,B 24.9609,C -1.444,E1 24.985,E2 185.1202} C_DIS
LIN {X -16.8577,Y -118.5811,Z 128,A -101.9362,B 24.9607,C -1.4493,E1 24.9767,E2 188.146} C_DIS
LIN {X -21.21,Y -117.8804,Z 128,A -103.8782,B 24.9602,C -1.4575,E1 24.9714,E2 190.0704} C_DIS
LIN {X -23.9783,Y -117.3487,Z 128,A -105.3615,B 24.9605,C -1.4519,E1 24.9672,E2 191.5686} C_DIS
LIN {X -27.1696,Y -116.6513,Z 128,A -106.9395,B 24.9605,C -1.4519,E1 24.9629,E2 193.1484} C_DIS
LIN {X -30.1149,Y -115.926,Z 128,A -108.5093,B 24.9608,C -1.4475,E1 24.9587,E2 194.7312} C_DIS
LIN {X -34.2422,Y -114.7744,Z 128,A -111.144,B 24.9621,C -1.4228,E1 24.9514,E2 197.4288} C_DIS
LIN {X -38.9413,Y -113.2679,Z 128,A -112.7459,B 24.9601,C -1.4585,E1 24.9474,E2 198.9489} C_DIS
LIN {X -41.1813,Y -112.4712,Z 128,A -113.954,B 24.9603,C -1.4564,E1 24.9442,E2 200.1645} C_DIS
LIN {X -44.7076,Y -111.1176,Z 128,A -115.762,B 24.9602,C -1.4581,E1 24.9395,E2 201.9723} C_DIS
LIN {X -48.9701,Y -109.3053,Z 128,A -117.9463,B 24.96,C -1.4619,E1 24.9339,E2 204.1527} C_DIS
LIN {X -51.8885,Y -107.9502,Z 128,A -119.5074,B 24.96,C -1.4628,E1 24.93,E2 205.7157} C_DIS
LIN {X -54.8757,Y -106.4635,Z 128,A -121.0759,B 24.9597,C -1.466,E1 24.9261,E2 207.2807} C_DIS
LIN {X -57.4807,Y -105.08,Z 128,A -122.4903,B 24.9597,C -1.4678,E1 24.9226,E2 208.695} C_DIS
LIN {X -60.2964,Y -103.4916,Z 128,A -124.2131,B 24.9599,C -1.4622,E1 24.9184,E2 210.4361} C_DIS
LIN {X -63.494,Y -101.5587,Z 128,A -125.8264,B 24.9594,C -1.4726,E1 24.9146,E2 212.0298} C_DIS
LIN {X -66.0519,Y -99.9141,Z 128,A -127.3708,B 24.9594,C -1.4709,E1 24.911,E2 213.583} C_DIS
LIN {X -71.2534,Y -96.2755,Z 128,A -130.3193,B 24.959,C -1.4799,E1 24.9043,E2 216.5203} C_DIS
LIN {X -74.8457,Y -93.5109,Z 128,A -132.9689,B 24.9599,C -1.463,E1 24.8983,E2 219.2201} C_DIS
LIN {X -77.4352,Y -91.3758,Z 128,A -133.9633,B 24.9583,C -1.4926,E1 24.8964,E2 220.1476} C_DIS
LIN {X -80.7652,Y -88.4462,Z 128,A -136.4507,B 24.9589,C -1.481,E1 24.8911,E2 222.6727} C_DIS
LIN {X -83.3386,Y -86.0257,Z 128,A -138.0323,B 24.9585,C -1.4892,E1 24.8879,E2 224.2413} C_DIS
LIN {X -85.4748,Y -83.9039,Z 128,A -139.431,B 24.9582,C -1.4941,E1 24.8852,E2 225.6342} C_DIS
LIN {X -88.3973,Y -80.8184,Z 128,A -141.5185,B 24.9581,C -1.4963,E1 24.8812,E2 227.7256} C_DIS
LIN {X -91.3738,Y -77.4376,Z 128,A -143.7581,B 24.958,C -1.4977,E1 24.8771,E2 229.9722} C_DIS
LIN {X -94.0095,Y -74.2151,Z 128,A -146.4857,B 24.9595,C -1.4711,E1 24.8722,E2 232.7757} C_DIS
LIN {X -97.2759,Y -69.88,Z 128,A -148.0903,B 24.9567,C -1.5198,E1 24.8697,E2 234.2721} C_DIS
LIN {X -100.483,Y -65.1856,Z 128,A -150.9093,B 24.9566,C -1.5225,E1 24.8653,E2 237.0987} C_DIS
LIN {X -103.1002,Y -60.959,Z 128,A -154.1053,B 24.9582,C -1.4943,E1 24.8606,E2 240.3785} C_DIS
LIN {X -105.5098,Y -56.6883,Z 128,A -155.7354,B 24.9561,C -1.5309,E1 24.8585,E2 241.9298} C_DIS
LIN {X -107.0471,Y -53.7301,Z 128,A -157.4848,B 24.9562,C -1.5289,E1 24.8563,E2 243.6936} C_DIS
LIN {X -109.2775,Y -49.0318,Z 128,A -159.888,B 24.9556,C -1.5396,E1 24.8534,E2 246.0843} C_DIS
LIN {X -110.8627,Y -45.3339,Z 128,A -161.8088,B 24.9553,C -1.5454,E1 24.8514,E2 248.0019} C_DIS
LIN {X -111.9795,Y -42.5001,Z 128,A -163.8582,B 24.9564,C -1.5248,E1 24.8493,E2 250.1118} C_DIS
LIN {X -113.4389,Y -38.4357,Z 128,A -165.0764,B 24.954,C -1.5667,E1 24.8483,E2 251.2372} C_DIS
LIN {X -114.4775,Y -35.2224,Z 128,A -167.5217,B 24.9558,C -1.5367,E1 24.8461,E2 253.768} C_DIS
LIN {X -115.6175,Y -31.2769,Z 128,A -169.4073,B 24.9552,C -1.5461,E1 24.8448,E2 255.6422} C_DIS
LIN {X -116.5545,Y -27.5882,Z 128,A -170.7167,B 24.9536,C -1.5732,E1 24.8439,E2 256.8947} C_DIS
LIN {X -117.4929,Y -23.2691,Z 128,A -173.1464,B 24.954,C -1.5666,E1 24.8425,E2 259.3544} C_DIS
LIN {X -118.1939,Y -19.3903,Z 128,A -174.9138,B 24.9534,C -1.5775,E1 24.8417,E2 261.1062} C_DIS
LIN {X -118.8043,Y -15.2062,Z 128,A -176.8379,B 24.9527,C -1.5882,E1 24.841,E2 263.0165} C_DIS
LIN {X -119.2142,Y -11.5741,Z 128,A -178.7071,B 24.9527,C -1.5887,E1 24.8404,E2 264.8955} C_DIS
LIN {X -119.5081,Y -7.9673,Z 128,A 179.6342,B 24.9522,C -1.5974,E1 24.8401,E2 266.5436} C_DIS
LIN {X -119.6935,Y -4.4313,Z 128,A 177.7867,B 24.9522,C -1.5964,E1 24.8398,E2 268.4045} C_DIS
LIN {X -119.7715,Y -0.7113,Z 128,A 176.1473,B 24.9515,C -1.6081,E1 24.8398,E2 270.0258} C_DIS
LIN {X -119.7395,Y 2.9394,Z 128,A 174.2472,B 24.9515,C -1.6074,E1 24.8398,E2 271.9392} C_DIS
LIN {X -119.5882,Y 6.658,Z 128,A 172.6164,B 24.9509,C -1.6195,E1 24.8401,E2 273.5509} C_DIS
LIN {X -119.3964,Y 9.4953,Z 128,A 171.1976,B 24.9507,C -1.6215,E1 24.8404,E2 274.9734} C_DIS
LIN {X -119.0556,Y 13.1085,Z 128,A 169.5057,B 24.9503,C -1.629,E1 24.8409,E2 276.6576} C_DIS
LIN {X -118.6174,Y 16.602,Z 128,A 167.765,B 24.9501,C -1.6322,E1 24.8415,E2 278.4012} C_DIS
LIN {X -118.0738,Y 20.1088,Z 128,A 166.1081,B 24.9496,C -1.6394,E1 24.8422,E2 280.0508} C_DIS
LIN {X -117.4101,Y 23.6789,Z 128,A 164.2977,B 24.9495,C -1.642,E1 24.8432,E2 281.8657} C_DIS
LIN {X -116.6848,Y 27.0243,Z 128,A 162.6276,B 24.9492,C -1.6459,E1 24.8442,E2 283.5363} C_DIS
LIN {X -114.996,Y 33.4951,Z 128,A 159.544,B 24.9483,C -1.6609,E1 24.8464,E2 286.6019} C_DIS
LIN {X -111.9959,Y 42.4568,Z 128,A 155.267,B 24.9468,C -1.6854,E1 24.8502,E2 290.8449} C_DIS
LIN {X -111.0483,Y 44.8777,Z 128,A 153.5805,B 24.9477,C -1.6707,E1 24.852,E2 292.5759} C_DIS
LIN {X -109.4839,Y 48.5738,Z 128,A 151.0436,B 24.9489,C -1.6509,E1 24.8549,E2 295.1741} C_DIS
LIN {X -107.5212,Y 52.7738,Z 128,A 149.6287,B 24.9464,C -1.6911,E1 24.8565,E2 296.5008} C_DIS
LIN {X -105.6106,Y 56.4999,Z 128,A 147.0311,B 24.9476,C -1.6722,E1 24.86,E2 299.1573} C_DIS
LIN {X -103.8837,Y 59.6141,Z 128,A 145.4135,B 24.9471,C -1.6808,E1 24.8622,E2 300.7628} C_DIS
LIN {X -102.0046,Y 62.7787,Z 128,A 143.8214,B 24.9463,C -1.6929,E1 24.8645,E2 302.3344} C_DIS
LIN {X -99.8951,Y 66.0806,Z 128,A 141.7834,B 24.9463,C -1.6914,E1 24.8676,E2 304.3862} C_DIS
LIN {X -97.1322,Y 70.0813,Z 128,A 139.2201,B 24.9466,C -1.6879,E1 24.8718,E2 306.9703} C_DIS
LIN {X -94.7511,Y 73.2662,Z 128,A 138.278,B 24.9437,C -1.7335,E1 24.8732,E2 307.8082} C_DIS
LIN {X -93.1157,Y 75.3335,Z 128,A 136.0475,B 24.9461,C -1.6959,E1 24.8773,E2 310.1387} C_DIS
LIN {X -90.5023,Y 78.455,Z 128,A 134.5428,B 24.9446,C -1.7196,E1 24.8799,E2 311.5937} C_DIS
LIN {X -87.0741,Y 82.2424,Z 128,A 132.0499,B 24.9443,C -1.7237,E1 24.8846,E2 314.0878} C_DIS
LIN {X -82.6145,Y 86.7235,Z 128,A 129.1605,B 24.9435,C -1.7368,E1 24.8903,E2 316.9584} C_DIS
LIN {X -80.5308,Y 88.6612,Z 128,A 127.4469,B 24.9442,C -1.725,E1 24.8939,E2 318.7068} C_DIS
LIN {X -77.4376,Y 91.3738,Z 128,A 125.762,B 24.9432,C -1.7416,E1 24.8974,E2 320.359} C_DIS
LIN {X -72.696,Y 95.1904,Z 128,A 122.8791,B 24.9427,C -1.7491,E1 24.9037,E2 323.2346} C_DIS
LIN {X -67.5626,Y 98.8999,Z 128,A 119.9362,B 24.942,C -1.7591,E1 24.9104,E2 326.164} C_DIS
LIN {X -64.1231,Y 101.165,Z 128,A 117.5357,B 24.943,C -1.7444,E1 24.9161,E2 328.6073} C_DIS
LIN {X -57.8762,Y 104.8635,Z 128,A 114.379,B 24.9417,C -1.7643,E1 24.9236,E2 331.7261} C_DIS
LIN {X -54.867,Y 106.468,Z 128,A 111.9625,B 24.9437,C -1.7333,E1 24.9298,E2 334.2228} C_DIS
LIN {X -50.3963,Y 108.6549,Z 128,A 110.3357,B 24.9413,C -1.7695,E1 24.9337,E2 335.7677} C_DIS
LIN {X -47.3417,Y 110.0216,Z 128,A 108.6828,B 24.9413,C -1.7695,E1 24.938,E2 337.4242} C_DIS
LIN {X -40.3058,Y 112.7899,Z 128,A 104.9873,B 24.9413,C -1.771,E1 24.9476,E2 341.1242} C_DIS
LIN {X -36.8933,Y 113.9497,Z 128,A 103.3196,B 24.9409,C -1.7756,E1 24.952,E2 342.7841} C_DIS
LIN {X -33.2415,Y 115.0697,Z 128,A 101.2694,B 24.9414,C -1.7679,E1 24.9575,E2 344.8561} C_DIS
LIN {X -29.5112,Y 116.0812,Z 128,A 99.7006,B 24.9405,C -1.7821,E1 24.9617,E2 346.3936} C_DIS
LIN {X -26.8497,Y 116.7252,Z 128,A 98.3556,B 24.9405,C -1.7818,E1 24.9654,E2 347.7411} C_DIS
LIN {X -23.5695,Y 117.4326,Z 128,A 96.667,B 24.9407,C -1.7794,E1 24.97,E2 349.4371} C_DIS
LIN {X -18.7227,Y 118.3017,Z 128,A 94.5466,B 24.9398,C -1.7916,E1 24.9758,E2 351.5308} C_DIS
Enddeposition()
END
